(* LS UPPER TRAILING DOT 4 PHASE WINDOW *)
ls_trailing_lower_dot_4_on_comp := ls_trailing_lower_dot_4_on + less_glue_strip_deg;
ls_trailing_lower_dot_4_off_comp := ls_trailing_lower_dot_4_off - less_glue_strip_deg;

phase_window_set_phases_data(
	begin_phase:=  ls_trailing_lower_dot_4_on_comp,
	end_phase:=  ls_trailing_lower_dot_4_off_comp,
	begin_delay:= 0,
	end_delay:= 0,
	begin_max_compensation:= 0,
	end_max_compensation:= 0,
	CONVERSION_this:= ls_trailing_lower_dot_4_phwin);	

(* LS UPPER TRAILING DOT 5 PHASE WINDOW *)
ls_trailing_lower_dot_5_on_comp := ls_trailing_lower_dot_5_on + less_glue_strip_deg;
ls_trailing_lower_dot_5_off_comp := ls_trailing_lower_dot_5_off - less_glue_strip_deg;

phase_window_set_phases_data(
	begin_phase:=  ls_trailing_lower_dot_5_on_comp,
	end_phase:=  ls_trailing_lower_dot_5_off_comp,
	begin_delay:= 0,
	end_delay:= 0,
	begin_max_compensation:= 0,
	end_max_compensation:= 0,
	CONVERSION_this:= ls_trailing_lower_dot_5_phwin);
	
(* LS UPPER TRAILING DOT 6 PHASE WINDOW *)
ls_trailing_lower_dot_6_on_comp := ls_trailing_lower_dot_6_on + less_glue_strip_deg;
ls_trailing_lower_dot_6_off_comp := ls_trailing_lower_dot_6_off - less_glue_strip_deg;

phase_window_set_phases_data(
	begin_phase:=  ls_trailing_lower_dot_6_on_comp,
	end_phase:=  ls_trailing_lower_dot_6_off_comp,
	begin_delay:= 0,
	end_delay:= 0,
	begin_max_compensation:= 0,
	end_max_compensation:= 0,
	CONVERSION_this:= ls_trailing_lower_dot_6_phwin);
END_ACTION

ACTION _handle_messages:
IF purge_command
THEN 
	process_message_set(errorID_1:= 1, errorID_2:= 0, errorID_3:= 0, CONVERSION_this:= purge_running);
ELSE
	process_message_reset(purge_running);
END_IF
END_ACTION

ACTION _handle_process_test:
;
END_ACTION

ACTION _mode_manager:
IF process_mode_req_is_pending(prc)
THEN
    process_apply_mode_req_first_step(prc);
    CASE process_get_mode(prc) OF
        MODE_TO_ABSENT:
			;
        MODE_TO_INACTIVE:
			;
        MODE_TO_TEST:
			;
        MODE_TO_OPERATIONAL:
			;
    END_CASE
    process_apply_mode_req_second_step(prc);
END_IF
END_ACTION

ACTION _object_manager:
IF objects_initialization()
THEN
	sub_process_init(
		object_name					:= 'csp_case_glue.prc', 
		process						:= csp_case.prc, 
		CONVERSION_this				:= prc);
		
	prc_path 						:= process_get_path(prc);
	
	process_message_init(
		object_name:= CONCAT(prc_path, '_purge_running'), 
		behaviour:= MESSAGE_BEHAVIOUR_STATE, 
		reset_timeout:= 0, 
		disableable:= FALSE, 
		individual_reset:= FALSE, 
		machine_reaction:= MACHINE_REACTION_STOP_IN_PHASE_ONE, 
		typology:= MESSAGE_TYPOLOGY_ABNORMAL, 
		process:= prc, 
		CONVERSION_this:= purge_running);
	
	//PRS 7/14/2021	
	process_message_init(
        object_name:= CONCAT(prc_path, '_OS_lower_glue_gun_disabled_wem'),
        behaviour:= MESSAGE_BEHAVIOUR_STATE,
        reset_timeout:= 0,
        disableable:= TRUE,
        individual_reset:= FALSE,
        machine_reaction:= MACHINE_REACTION_NO_STOP, 
        typology:=  MESSAGE_TYPOLOGY_NORMAL, 
        process:= prc,
        CONVERSION_this:= OS_lower_glue_gun_disabled_wem);
	
	//PRS 7/14/2021	
	process_message_init(
        object_name:= CONCAT(prc_path, '_OS_upper_glue_gun_disabled_wem'),
        behaviour:= MESSAGE_BEHAVIOUR_STATE,
        reset_timeout:= 0,
        disableable:= TRUE,
        individual_reset:= FALSE,
        machine_reaction:= MACHINE_REACTION_NO_STOP, 
        typology:=  MESSAGE_TYPOLOGY_NORMAL, 
        process:= prc,
        CONVERSION_this:= OS_upper_glue_gun_disabled_wem);	

	//PRS 7/14/2021	
	process_message_init(
        object_name:= CONCAT(prc_path, '_LS_lower_glue_gun_disabled_wem'),
        behaviour:= MESSAGE_BEHAVIOUR_STATE,
        reset_timeout:= 0,
        disableable:= TRUE,
        individual_reset:= FALSE,
        machine_reaction:= MACHINE_REACTION_NO_STOP, 
        typology:=  MESSAGE_TYPOLOGY_NORMAL, 
        process:= prc,
        CONVERSION_this:= LS_lower_glue_gun_disabled_wem);
	
	//PRS 7/14/2021	
	process_message_init(
        object_name:= CONCAT(prc_path, '_LS_upper_glue_gun_disabled_wem'),
        behaviour:= MESSAGE_BEHAVIOUR_STATE,
        reset_timeout:= 0,
        disableable:= TRUE,
        individual_reset:= FALSE,
        machine_reaction:= MACHINE_REACTION_NO_STOP, 
        typology:=  MESSAGE_TYPOLOGY_NORMAL, 
        process:= prc,
        CONVERSION_this:= LS_upper_glue_gun_disabled_wem);		
		
		
	motorization_conditioner_init(
		object_name					:=	CONCAT(prc_path, '_purge_active_motcond'),
		velocity_limit				:=	0.0,
		velocity_limit_active		:=	FALSE,
		idle_handshake_active		:=	FALSE,
		execute_handshake_active	:=	TRUE,
		hold_handshake_active		:=	FALSE,
		suspend_handshake_active	:=	FALSE,
		complete_handshake_active	:=	FALSE,
		abort_handshake_active		:=	FALSE,
		stop_handshake_active		:=	FALSE,
		origin						:=	MOTORIZATION_CONDITIONER_ORIGIN_INTERNAL,
		manager						:=	csp_main_motorization_manager.motm,
		process						:=	prc,
		CONVERSION_this				:=	purge_active_motcond);

		
	command_button_init(
	    object_name 				:= CONCAT(prc_path, '_hmi_purge_active_cbtn'),
	    process 					:= prc,
	    CONVERSION_this 			:= hmi_purge_active_cbtn);
		
	hmi_graphic_object_status_init(
        object_name         		:= CONCAT(prc_path, '_hmi_purge_active_hgos'),
        process             		:= prc,
        CONVERSION_this             := hmi_purge_active_hgos);	
		
	hmi_graphic_object_status_init(
        object_name         		:= CONCAT(prc_path, '_hmi_glue_ready_hgos'),
        process             		:= prc,
        CONVERSION_this             := hmi_glue_ready_hgos);
		
	hmi_graphic_object_status_init(
        object_name         		:= CONCAT(prc_path, '_hmi_glue_not_ready_hgos'),
        process             		:= prc,
        CONVERSION_this             := hmi_glue_not_ready_hgos);	
	
//Glue Purge pb OS upper gun 1
	command_button_init(
	    object_name 				:= CONCAT(prc_path, '_hmi_os_glue_upper_gun1_cbtn'),
	    process 					:= prc,
	    CONVERSION_this 			:= hmi_os_glue_upper_gun1_cbtn);
		
	hmi_graphic_object_status_init(
        object_name         		:= CONCAT(prc_path, '_hmi_os_glue_upper_gun1_hgos'),
        process             		:= prc,
        CONVERSION_this             := hmi_os_glue_upper_gun1_hgos);	

//Glue Purge pb OS upper gun 2
	command_button_init(
	    object_name 				:= CONCAT(prc_path, '_hmi_os_glue_upper_gun2_cbtn'),
	    process 					:= prc,
	    CONVERSION_this 			:= hmi_os_glue_upper_gun2_cbtn);
		
	hmi_graphic_object_status_init(
        object_name         		:= CONCAT(prc_path, '_hmi_os_glue_upper_gun2_hgos'),
        process             		:= prc,
        CONVERSION_this             := hmi_os_glue_upper_gun2_hgos);			

//Glue Purge pb OS lower gun 1
	command_button_init(
	    object_name 				:= CONCAT(prc_path, '_hmi_os_glue_lower_gun1_cbtn'),
	    process 					:= prc,
	    CONVERSION_this 			:= hmi_os_glue_lower_gun1_cbtn);
		
	hmi_graphic_object_status_init(
        object_name         		:= CONCAT(prc_path, '_hmi_os_glue_lower_gun1_hgos'),
        process             		:= prc,
        CONVERSION_this             := hmi_os_glue_lower_gun1_hgos);	

//Glue Purge pb OS lower gun 2
	command_button_init(
	    object_name 				:= CONCAT(prc_path, '_hmi_os_glue_lower_gun2_cbtn'),
	    process 					:= prc,
	    CONVERSION_this 			:= hmi_os_glue_lower_gun2_cbtn);
		
	hmi_graphic_object_status_init(
        object_name         		:= CONCAT(prc_path, '_hmi_os_glue_lower_gun2_hgos'),
        process             		:= prc,
        CONVERSION_this             := hmi_os_glue_lower_gun2_hgos);	


//Glue Purge pb LS upper gun 1
	command_button_init(
	    object_name 				:= CONCAT(prc_path, '_hmi_ls_glue_upper_gun1_cbtn'),
	    process 					:= prc,
	    CONVERSION_this 			:= hmi_ls_glue_upper_gun1_cbtn);
		
	hmi_graphic_object_status_init(
        object_name         		:= CONCAT(prc_path, '_hmi_ls_glue_upper_gun1_hgos'),
        process             		:= prc,
        CONVERSION_this             := hmi_ls_glue_upper_gun1_hgos);	

//Glue Purge pb LS upper gun 2
	command_button_init(
	    object_name 				:= CONCAT(prc_path, '_hmi_ls_glue_upper_gun2_cbtn'),
	    process 					:= prc,
	    CONVERSION_this 			:= hmi_ls_glue_upper_gun2_cbtn);
		
	hmi_graphic_object_status_init(
        object_name         		:= CONCAT(prc_path, '_hmi_ls_glue_upper_gun2_hgos'),
        process             		:= prc,
        CONVERSION_this             := hmi_ls_glue_upper_gun2_hgos);			

//Glue Purge pb LS lower gun 1
	command_button_init(
	    object_name 				:= CONCAT(prc_path, '_hmi_Ls_glue_lower_gun1_cbtn'),
	    process 					:= prc,
	    CONVERSION_this 			:= hmi_ls_glue_lower_gun1_cbtn);
		
	hmi_graphic_object_status_init(
        object_name         		:= CONCAT(prc_path, '_hmi_ls_glue_lower_gun1_hgos'),
        process             		:= prc,
        CONVERSION_this             := hmi_ls_glue_lower_gun1_hgos);	

//Glue Purge pb LS lower gun 2
	command_button_init(
	    object_name 				:= CONCAT(prc_path, '_hmi_ls_glue_lower_gun2_cbtn'),
	    process 					:= prc,
	    CONVERSION_this 			:= hmi_ls_glue_lower_gun2_cbtn);
		
	hmi_graphic_object_status_init(
        object_name         		:= CONCAT(prc_path, '_hmi_ls_glue_lower_gun2_hgos'),
        process             		:= prc,
        CONVERSION_this             := hmi_ls_glue_lower_gun2_hgos);

	//Created to be the axis for the shift registers	
	phase_generator_init(
		object_name								:=CONCAT(PRC_PATH, '_glue_vm_phgen'), 
		modulo									:=360 , 
		resolution								:= PHASE_GENERATOR_RESOLUTION_UNIT, 
		axis									:= csp_case_transport_os_trailing.axis, 
		process									:=prc , 
		CONVERSION_this							:= glue_vm_phgen);

//Upper major flap check cam and phase generator		

	phase_window_init(
		object_name								:=CONCAT(PRC_PATH, '_glue_phwin'), 
		begin_phase								:=glue_leading_upper_on, 
		end_phase								:=glue_leading_upper_off, 
		begin_delay								:=0, 
		end_delay								:=0, 
		begin_max_compensation					:=0, 
		end_max_compensation					:=0, 
		generator								:=glue_vm_phgen , 
		process									:=prc , 
		CONVERSION_this							:=glue_leading_upper_phwin);	
		
//lower major flap check cam and phase generator 		

	phase_window_init(
		object_name								:=CONCAT(PRC_PATH, '_glue_phwin'), 
		begin_phase								:=glue_leading_lower_on, 
		end_phase								:=glue_leading_lower_off, 
		begin_delay								:=0, 
		end_delay								:=0, 
		begin_max_compensation					:=0, 
		end_max_compensation					:=0, 
		generator								:=glue_vm_phgen , 
		process									:=prc , 
		CONVERSION_this							:=glue_leading_lower_phwin);	

//Upper major flap check 2 cam and phase generator		
	
	phase_window_init(
		object_name								:=CONCAT(PRC_PATH, '_glue_2_phwin'), 
		begin_phase								:=glue_trailing_upper_on, 
		end_phase								:=glue_trailing_upper_off, 
		begin_delay								:=0, 
		end_delay								:=0, 
		begin_max_compensation					:=0, 
		end_max_compensation					:=0, 
		generator								:=glue_vm_phgen , 
		process									:=prc , 
		CONVERSION_this							:=glue_trailing_upper_phwin);	
		
//Lower major flap check 2 cam and phase generator		
	
	phase_window_init(
		object_name								:=CONCAT(PRC_PATH, '_glue_2_phwin'), 
		begin_phase								:=glue_trailing_lower_on, 
		end_phase								:=glue_trailing_lower_off, 
		begin_delay								:=0, 
		end_delay								:=0, 
		begin_max_compensation					:=0, 
		end_max_compensation					:=0, 
		generator								:=glue_vm_phgen , 
		process									:=prc , 
		CONVERSION_this							:=glue_trailing_lower_phwin);	
		
		
		
	(* NEW GLUE GUNS USING DIGITAL OUTPUTS *)
	digital_output_init(
		object_name 			:= CONCAT(prc_path, '_os_upper_gun_1_do'),
		polarity_direct 		:= TRUE,
		process 				:= prc,
		CONVERSION_this 		:= os_upper_gun_1_do);
		
	digital_output_init(
		object_name 			:= CONCAT(prc_path, '_os_upper_gun_2_do'),
		polarity_direct 		:= TRUE,
		process 				:= prc,
		CONVERSION_this 		:= os_upper_gun_2_do);
		
	digital_output_init(
		object_name 			:= CONCAT(prc_path, '_os_lower_gun_1_do'),
		polarity_direct 		:= TRUE,
		process 				:= prc,
		CONVERSION_this 		:= os_lower_gun_1_do);
		
	digital_output_init(
		object_name 			:= CONCAT(prc_path, '_os_lower_gun_2_do'),
		polarity_direct 		:= TRUE,
		process 				:= prc,
		CONVERSION_this 		:= os_lower_gun_2_do);
		
	digital_output_init(
		object_name 			:= CONCAT(prc_path, '_ls_upper_gun_1_do'),
		polarity_direct 		:= TRUE,
		process 				:= prc,
		CONVERSION_this 		:= ls_upper_gun_1_do);
		
	digital_output_init(
		object_name 			:= CONCAT(prc_path, '_ls_upper_gun_2_do'),
		polarity_direct 		:= TRUE,
		process 				:= prc,
		CONVERSION_this 		:= ls_upper_gun_2_do);
		
	digital_output_init(
		object_name 			:= CONCAT(prc_path, '_ls_lower_gun_1_do'),
		polarity_direct 		:= TRUE,
		process 				:= prc,
		CONVERSION_this 		:= ls_lower_gun_1_do);
		
	digital_output_init(
		object_name 			:= CONCAT(prc_path, '_ls_lower_gun_2_do'),
		polarity_direct 		:= TRUE,
		process 				:= prc,
		CONVERSION_this 		:= ls_lower_gun_2_do);
		
	(* OS LEADING UPPER PHWIN *)
	phase_window_init(
		object_name								:= CONCAT(PRC_PATH, '_os_leading_upper_dot_1_phwin'), 
		begin_phase								:= 0, // SET AT RUNTIME
		end_phase								:= 0, // SET AT RUNTIME
		begin_delay								:= 0, 
		end_delay								:= 0, 
		begin_max_compensation					:= 0, 
		end_max_compensation					:= 0, 
		generator								:= glue_vm_phgen , 
		process									:= prc , 
		CONVERSION_this							:= os_leading_upper_dot_1_phwin);	
		
	phase_window_init(
		object_name								:= CONCAT(PRC_PATH, '_os_leading_upper_dot_2_phwin'), 
		begin_phase								:= 0, // SET AT RUNTIME
		end_phase								:= 0, // SET AT RUNTIME
		begin_delay								:= 0, 
		end_delay								:= 0, 
		begin_max_compensation					:= 0, 
		end_max_compensation					:= 0, 
		generator								:= glue_vm_phgen , 
		process									:= prc , 
		CONVERSION_this							:= os_leading_upper_dot_2_phwin);	
		
	phase_window_init(
		object_name								:= CONCAT(PRC_PATH, '_os_leading_upper_dot_3_phwin'), 
		begin_phase								:= 0, // SET AT RUNTIME
		end_phase								:= 0, // SET AT RUNTIME
		begin_delay								:= 0, 
		end_delay								:= 0, 
		begin_max_compensation					:= 0, 
		end_max_compensation					:= 0, 
		generator								:= glue_vm_phgen , 
		process									:= prc , 
		CONVERSION_this							:= os_leading_upper_dot_3_phwin);	
		
	phase_window_init(
		object_name								:= CONCAT(PRC_PATH, '_os_leading_upper_dot_4_phwin'), 
		begin_phase								:= 0, // SET AT RUNTIME
		end_phase								:= 0, // SET AT RUNTIME
		begin_delay								:= 0, 
		end_delay								:= 0, 
		begin_max_compensation					:= 0, 
		end_max_compensation					:= 0, 
		generator								:= glue_vm_phgen , 
		process									:= prc , 
		CONVERSION_this							:= os_leading_upper_dot_4_phwin);	
		
	phase_window_init(
		object_name								:= CONCAT(PRC_PATH, '_os_leading_upper_dot_5_phwin'), 
		begin_phase								:= 0, // SET AT RUNTIME
		end_phase								:= 0, // SET AT RUNTIME
		begin_delay								:= 0, 
		end_delay								:= 0, 
		begin_max_compensation					:= 0, 
		end_max_compensation					:= 0, 
		generator								:= glue_vm_phgen , 
		process									:= prc , 
		CONVERSION_this							:= os_leading_upper_dot_5_phwin);	
		
	phase_window_init(
		object_name								:= CONCAT(PRC_PATH, '_os_leading_upper_dot_6_phwin'), 
		begin_phase								:= 0, // SET AT RUNTIME
		end_phase								:= 0, // SET AT RUNTIME
		begin_delay								:= 0, 
		end_delay								:= 0, 
		begin_max_compensation					:= 0, 
		end_max_compensation					:= 0, 
		generator								:= glue_vm_phgen , 
		process									:= prc , 
		CONVERSION_this							:= os_leading_upper_dot_6_phwin);
		
		
	(* OS LEADING LOWER PHWIN *)
	phase_window_init(
		object_name								:= CONCAT(PRC_PATH, '_os_leading_lower_dot_1_phwin'), 
		begin_phase								:= 0, // SET AT RUNTIME
		end_phase								:= 0, // SET AT RUNTIME
		begin_delay								:= 0, 
		end_delay								:= 0, 
		begin_max_compensation					:= 0, 
		end_max_compensation					:= 0, 
		generator								:= glue_vm_phgen , 
		process									:= prc , 
		CONVERSION_this							:= os_leading_lower_dot_1_phwin);	
		
	phase_window_init(
		object_name								:= CONCAT(PRC_PATH, '_os_leading_lower_dot_2_phwin'), 
		begin_phase								:= 0, // SET AT RUNTIME
		end_phase								:= 0, // SET AT RUNTIME
		begin_delay								:= 0, 
		end_delay								:= 0, 
		begin_max_compensation					:= 0, 
		end_max_compensation					:= 0, 
		generator								:= glue_vm_phgen , 
		process									:= prc , 
		CONVERSION_this							:= os_leading_lower_dot_2_phwin);	
		
	phase_window_init(
		object_name								:= CONCAT(PRC_PATH, '_os_leading_lower_dot_3_phwin'), 
		begin_phase								:= 0, // SET AT RUNTIME
		end_phase								:= 0, // SET AT RUNTIME
		begin_delay								:= 0, 
		end_delay								:= 0, 
		begin_max_compensation					:= 0, 
		end_max_compensation					:= 0, 
		generator								:= glue_vm_phgen , 
		process									:= prc , 
		CONVERSION_this							:= os_leading_lower_dot_3_phwin);	
		
	phase_window_init(
		object_name								:= CONCAT(PRC_PATH, '_os_leading_lower_dot_4_phwin'), 
		begin_phase								:= 0, // SET AT RUNTIME
		end_phase								:= 0, // SET AT RUNTIME
		begin_delay								:= 0, 
		end_delay								:= 0, 
		begin_max_compensation					:= 0, 
		end_max_compensation					:= 0, 
		generator								:= glue_vm_phgen , 
		process									:= prc , 
		CONVERSION_this							:= os_leading_lower_dot_4_phwin);	
		
	phase_window_init(
		object_name								:= CONCAT(PRC_PATH, '_os_leading_lower_dot_5_phwin'), 
		begin_phase								:= 0, // SET AT RUNTIME
		end_phase								:= 0, // SET AT RUNTIME
		begin_delay								:= 0, 
		end_delay								:= 0, 
		begin_max_compensation					:= 0, 
		end_max_compensation					:= 0, 
		generator								:= glue_vm_phgen , 
		process									:= prc , 
		CONVERSION_this							:= os_leading_lower_dot_5_phwin);	
		
	phase_window_init(
		object_name								:= CONCAT(PRC_PATH, '_os_leading_lower_dot_6_phwin'), 
		begin_phase								:= 0, // SET AT RUNTIME
		end_phase								:= 0, // SET AT RUNTIME
		begin_delay								:= 0, 
		end_delay								:= 0, 
		begin_max_compensation					:= 0, 
		end_max_compensation					:= 0, 
		generator								:= glue_vm_phgen , 
		process									:= prc , 
		CONVERSION_this							:= os_leading_lower_dot_6_phwin);	
		
	(* OS trailing UPPER PHWIN *)
	phase_window_init(
		object_name								:= CONCAT(PRC_PATH, '_os_trailing_upper_dot_1_phwin'), 
		begin_phase								:= 0, // SET AT RUNTIME
		end_phase								:= 0, // SET AT RUNTIME
		begin_delay								:= 0, 
		end_delay								:= 0, 
		begin_max_compensation					:= 0, 
		end_max_compensation					:= 0, 
		generator								:= glue_vm_phgen , 
		process									:= prc , 
		CONVERSION_this							:= os_trailing_upper_dot_1_phwin);	
		
	phase_window_init(
		object_name								:= CONCAT(PRC_PATH, '_os_trailing_upper_dot_2_phwin'), 
		begin_phase								:= 0, // SET AT RUNTIME
		end_phase								:= 0, // SET AT RUNTIME
		begin_delay								:= 0, 
		end_delay								:= 0, 
		begin_max_compensation					:= 0, 
		end_max_compensation					:= 0, 
		generator								:= glue_vm_phgen , 
		process									:= prc , 
		CONVERSION_this							:= os_trailing_upper_dot_2_phwin);	
		
	phase_window_init(
		object_name								:= CONCAT(PRC_PATH, '_os_trailing_upper_dot_3_phwin'), 
		begin_phase								:= 0, // SET AT RUNTIME
		end_phase								:= 0, // SET AT RUNTIME
		begin_delay								:= 0, 
		end_delay								:= 0, 
		begin_max_compensation					:= 0, 
		end_max_compensation					:= 0, 
		generator								:= glue_vm_phgen , 
		process									:= prc , 
		CONVERSION_this							:= os_trailing_upper_dot_3_phwin);	
		
	phase_window_init(
		object_name								:= CONCAT(PRC_PATH, '_os_trailing_upper_dot_4_phwin'), 
		begin_phase								:= 0, // SET AT RUNTIME
		end_phase								:= 0, // SET AT RUNTIME
		begin_delay								:= 0, 
		end_delay								:= 0, 
		begin_max_compensation					:= 0, 
		end_max_compensation					:= 0, 
		generator								:= glue_vm_phgen , 
		process									:= prc , 
		CONVERSION_this							:= os_trailing_upper_dot_4_phwin);	
		
	phase_window_init(
		object_name								:= CONCAT(PRC_PATH, '_os_trailing_upper_dot_5_phwin'), 
		begin_phase								:= 0, // SET AT RUNTIME
		end_phase								:= 0, // SET AT RUNTIME
		begin_delay								:= 0, 
		end_delay								:= 0, 
		begin_max_compensation					:= 0, 
		end_max_compensation					:= 0, 
		generator								:= glue_vm_phgen , 
		process									:= prc , 
		CONVERSION_this							:= os_trailing_upper_dot_5_phwin);	
		
	phase_window_init(
		object_name								:= CONCAT(PRC_PATH, '_os_trailing_upper_dot_6_phwin'), 
		begin_phase								:= 0, // SET AT RUNTIME
		end_phase								:= 0, // SET AT RUNTIME
		begin_delay								:= 0, 
		end_delay								:= 0, 
		begin_max_compensation					:= 0, 
		end_max_compensation					:= 0, 
		generator								:= glue_vm_phgen , 
		process									:= prc , 
		CONVERSION_this							:= os_trailing_upper_dot_6_phwin);	
		
		
	(* OS trailing LOWER PHWIN *)
	phase_window_init(
		object_name								:= CONCAT(PRC_PATH, '_os_trailing_lower_dot_1_phwin'), 
		begin_phase								:= 0, // SET AT RUNTIME
		end_phase								:= 0, // SET AT RUNTIME
		begin_delay								:= 0, 
		end_delay								:= 0, 
		begin_max_compensation					:= 0, 
		end_max_compensation					:= 0, 
		generator								:= glue_vm_phgen , 
		process									:= prc , 
		CONVERSION_this							:= os_trailing_lower_dot_1_phwin);	
		
	phase_window_init(
		object_name								:= CONCAT(PRC_PATH, '_os_trailing_lower_dot_2_phwin'), 
		begin_phase								:= 0, // SET AT RUNTIME
		end_phase								:= 0, // SET AT RUNTIME
		begin_delay								:= 0, 
		end_delay								:= 0, 
		begin_max_compensation					:= 0, 
		end_max_compensation					:= 0, 
		generator								:= glue_vm_phgen , 
		process									:= prc , 
		CONVERSION_this							:= os_trailing_lower_dot_2_phwin);	
		
	phase_window_init(
		object_name								:= CONCAT(PRC_PATH, '_os_trailing_lower_dot_3_phwin'), 
		begin_phase								:= 0, // SET AT RUNTIME
		end_phase								:= 0, // SET AT RUNTIME
		begin_delay								:= 0, 
		end_delay								:= 0, 
		begin_max_compensation					:= 0, 
		end_max_compensation					:= 0, 
		generator								:= glue_vm_phgen , 
		process									:= prc , 
		CONVERSION_this							:= os_trailing_lower_dot_3_phwin);	
		
	phase_window_init(
		object_name								:= CONCAT(PRC_PATH, '_os_trailing_lower_dot_4_phwin'), 
		begin_phase								:= 0, // SET AT RUNTIME
		end_phase								:= 0, // SET AT RUNTIME
		begin_delay								:= 0, 
		end_delay								:= 0, 
		begin_max_compensation					:= 0, 
		end_max_compensation					:= 0, 
		generator								:= glue_vm_phgen , 
		process									:= prc , 
		CONVERSION_this							:= os_trailing_lower_dot_4_phwin);
		
	phase_window_init(
		object_name								:= CONCAT(PRC_PATH, '_os_trailing_lower_dot_5_phwin'), 
		begin_phase								:= 0, // SET AT RUNTIME
		end_phase								:= 0, // SET AT RUNTIME
		begin_delay								:= 0, 
		end_delay								:= 0, 
		begin_max_compensation					:= 0, 
		end_max_compensation					:= 0, 
		generator								:= glue_vm_phgen , 
		process									:= prc , 
		CONVERSION_this							:= os_trailing_lower_dot_5_phwin);	
		
	phase_window_init(
		object_name								:= CONCAT(PRC_PATH, '_os_trailing_lower_dot_6_phwin'), 
		begin_phase								:= 0, // SET AT RUNTIME
		end_phase								:= 0, // SET AT RUNTIME
		begin_delay								:= 0, 
		end_delay								:= 0, 
		begin_max_compensation					:= 0, 
		end_max_compensation					:= 0, 
		generator								:= glue_vm_phgen , 
		process									:= prc , 
		CONVERSION_this							:= os_trailing_lower_dot_6_phwin);
		
	
	(* LS LEADING UPPER PHWIN *)
	phase_window_init(
		object_name								:= CONCAT(PRC_PATH, '_ls_leading_upper_dot_1_phwin'), 
		begin_phase								:= 0, // SET AT RUNTIME
		end_phase								:= 0, // SET AT RUNTIME
		begin_delay								:= 0, 
		end_delay								:= 0, 
		begin_max_compensation					:= 0, 
		end_max_compensation					:= 0, 
		generator								:= glue_vm_phgen , 
		process									:= prc , 
		CONVERSION_this							:= ls_leading_upper_dot_1_phwin);	
		
	phase_window_init(
		object_name								:= CONCAT(PRC_PATH, '_ls_leading_upper_dot_2_phwin'), 
		begin_phase								:= 0, // SET AT RUNTIME
		end_phase								:= 0, // SET AT RUNTIME
		begin_delay								:= 0, 
		end_delay								:= 0, 
		begin_max_compensation					:= 0, 
		end_max_compensation					:= 0, 
		generator								:= glue_vm_phgen , 
		process									:= prc , 
		CONVERSION_this							:= ls_leading_upper_dot_2_phwin);	
		
	phase_window_init(
		object_name								:= CONCAT(PRC_PATH, '_ls_leading_upper_dot_3_phwin'), 
		begin_phase								:= 0, // SET AT RUNTIME
		end_phase								:= 0, // SET AT RUNTIME
		begin_delay								:= 0, 
		end_delay								:= 0, 
		begin_max_compensation					:= 0, 
		end_max_compensation					:= 0, 
		generator								:= glue_vm_phgen , 
		process									:= prc , 
		CONVERSION_this							:= ls_leading_upper_dot_3_phwin);	
		
	phase_window_init(
		object_name								:= CONCAT(PRC_PATH, '_ls_leading_upper_dot_4_phwin'), 
		begin_phase								:= 0, // SET AT RUNTIME
		end_phase								:= 0, // SET AT RUNTIME
		begin_delay								:= 0, 
		end_delay								:= 0, 
		begin_max_compensation					:= 0, 
		end_max_compensation					:= 0, 
		generator								:= glue_vm_phgen , 
		process									:= prc , 
		CONVERSION_this							:= ls_leading_upper_dot_4_phwin);		
		
	phase_window_init(
		object_name								:= CONCAT(PRC_PATH, '_ls_leading_upper_dot_5_phwin'), 
		begin_phase								:= 0, // SET AT RUNTIME
		end_phase								:= 0, // SET AT RUNTIME
		begin_delay								:= 0, 
		end_delay								:= 0, 
		begin_max_compensation					:= 0, 
		end_max_compensation					:= 0, 
		generator								:= glue_vm_phgen , 
		process									:= prc , 
		CONVERSION_this							:= ls_leading_upper_dot_5_phwin);	
		
	phase_window_init(
		object_name								:= CONCAT(PRC_PATH, '_ls_leading_upper_dot_6_phwin'), 
		begin_phase								:= 0, // SET AT RUNTIME
		end_phase								:= 0, // SET AT RUNTIME
		begin_delay								:= 0, 
		end_delay								:= 0, 
		begin_max_compensation					:= 0, 
		end_max_compensation					:= 0, 
		generator								:= glue_vm_phgen , 
		process									:= prc , 
		CONVERSION_this							:= ls_leading_upper_dot_6_phwin);	
		
		
	(* LS LEADING LOWER PHWIN *)
	phase_window_init(
		object_name								:= CONCAT(PRC_PATH, '_ls_leading_lower_dot_1_phwin'), 
		begin_phase								:= 0, // SET AT RUNTIME
		end_phase								:= 0, // SET AT RUNTIME
		begin_delay								:= 0, 
		end_delay								:= 0, 
		begin_max_compensation					:= 0, 
		end_max_compensation					:= 0, 
		generator								:= glue_vm_phgen , 
		process									:= prc , 
		CONVERSION_this							:= ls_leading_lower_dot_1_phwin);	
		
	phase_window_init(
		object_name								:= CONCAT(PRC_PATH, '_ls_leading_lower_dot_2_phwin'), 
		begin_phase								:= 0, // SET AT RUNTIME
		end_phase								:= 0, // SET AT RUNTIME
		begin_delay								:= 0, 
		end_delay								:= 0, 
		begin_max_compensation					:= 0, 
		end_max_compensation					:= 0, 
		generator								:= glue_vm_phgen , 
		process									:= prc , 
		CONVERSION_this							:= ls_leading_lower_dot_2_phwin);	
		
	phase_window_init(
		object_name								:= CONCAT(PRC_PATH, '_ls_leading_lower_dot_3_phwin'), 
		begin_phase								:= 0, // SET AT RUNTIME
		end_phase								:= 0, // SET AT RUNTIME
		begin_delay								:= 0, 
		end_delay								:= 0, 
		begin_max_compensation					:= 0, 
		end_max_compensation					:= 0, 
		generator								:= glue_vm_phgen , 
		process									:= prc , 
		CONVERSION_this							:= ls_leading_lower_dot_3_phwin);	
		
	phase_window_init(
		object_name								:= CONCAT(PRC_PATH, '_ls_leading_lower_dot_4_phwin'), 
		begin_phase								:= 0, // SET AT RUNTIME
		end_phase								:= 0, // SET AT RUNTIME
		begin_delay								:= 0, 
		end_delay								:= 0, 
		begin_max_compensation					:= 0, 
		end_max_compensation					:= 0, 
		generator								:= glue_vm_phgen , 
		process									:= prc , 
		CONVERSION_this							:= ls_leading_lower_dot_4_phwin);		
		
	phase_window_init(
		object_name								:= CONCAT(PRC_PATH, '_ls_leading_lower_dot_5_phwin'), 
		begin_phase								:= 0, // SET AT RUNTIME
		end_phase								:= 0, // SET AT RUNTIME
		begin_delay								:= 0, 
		end_delay								:= 0, 
		begin_max_compensation					:= 0, 
		end_max_compensation					:= 0, 
		generator								:= glue_vm_phgen , 
		process									:= prc , 
		CONVERSION_this							:= ls_leading_lower_dot_5_phwin);	
		
	phase_window_init(
		object_name								:= CONCAT(PRC_PATH, '_ls_leading_lower_dot_6_phwin'), 
		begin_phase								:= 0, // SET AT RUNTIME
		end_phase								:= 0, // SET AT RUNTIME
		begin_delay								:= 0, 
		end_delay								:= 0, 
		begin_max_compensation					:= 0, 
		end_max_compensation					:= 0, 
		generator								:= glue_vm_phgen , 
		process									:= prc , 
		CONVERSION_this							:= ls_leading_lower_dot_6_phwin);	
		
	(* LS trailing UPPER PHWIN *)
	phase_window_init(
		object_name								:= CONCAT(PRC_PATH, '_ls_trailing_upper_dot_1_phwin'), 
		begin_phase								:= 0, // SET AT RUNTIME
		end_phase								:= 0, // SET AT RUNTIME
		begin_delay								:= 0, 
		end_delay								:= 0, 
		begin_max_compensation					:= 0, 
		end_max_compensation					:= 0, 
		generator								:= glue_vm_phgen , 
		process									:= prc , 
		CONVERSION_this							:= ls_trailing_upper_dot_1_phwin);	
		
	phase_window_init(
		object_name								:= CONCAT(PRC_PATH, '_ls_trailing_upper_dot_2_phwin'), 
		begin_phase								:= 0, // SET AT RUNTIME
		end_phase								:= 0, // SET AT RUNTIME
		begin_delay								:= 0, 
		end_delay								:= 0, 
		begin_max_compensation					:= 0, 
		end_max_compensation					:= 0, 
		generator								:= glue_vm_phgen , 
		process									:= prc , 
		CONVERSION_this							:= ls_trailing_upper_dot_2_phwin);	
		
	phase_window_init(
		object_name								:= CONCAT(PRC_PATH, '_ls_trailing_upper_dot_3_phwin'), 
		begin_phase								:= 0, // SET AT RUNTIME
		end_phase								:= 0, // SET AT RUNTIME
		begin_delay								:= 0, 
		end_delay								:= 0, 
		begin_max_compensation					:= 0, 
		end_max_compensation					:= 0, 
		generator								:= glue_vm_phgen , 
		process									:= prc , 
		CONVERSION_this							:= ls_trailing_upper_dot_3_phwin);	
		
	phase_window_init(
		object_name								:= CONCAT(PRC_PATH, '_ls_trailing_upper_dot_4_phwin'), 
		begin_phase								:= 0, // SET AT RUNTIME
		end_phase								:= 0, // SET AT RUNTIME
		begin_delay								:= 0, 
		end_delay								:= 0, 
		begin_max_compensation					:= 0, 
		end_max_compensation					:= 0, 
		generator								:= glue_vm_phgen , 
		process									:= prc , 
		CONVERSION_this							:= ls_trailing_upper_dot_4_phwin);	
		
	phase_window_init(
		object_name								:= CONCAT(PRC_PATH, '_ls_trailing_upper_dot_3_phwin'), 
		begin_phase								:= 0, // SET AT RUNTIME
		end_phase								:= 0, // SET AT RUNTIME
		begin_delay								:= 0, 
		end_delay								:= 0, 
		begin_max_compensation					:= 0, 
		end_max_compensation					:= 0, 
		generator								:= glue_vm_phgen , 
		process									:= prc , 
		CONVERSION_this							:= ls_trailing_upper_dot_5_phwin);	
		
	phase_window_init(
		object_name								:= CONCAT(PRC_PATH, '_ls_trailing_upper_dot_4_phwin'), 
		begin_phase								:= 0, // SET AT RUNTIME
		end_phase								:= 0, // SET AT RUNTIME
		begin_delay								:= 0, 
		end_delay								:= 0, 
		begin_max_compensation					:= 0, 
		end_max_compensation					:= 0, 
		generator								:= glue_vm_phgen , 
		process									:= prc , 
		CONVERSION_this							:= ls_trailing_upper_dot_6_phwin);	
		
		
	(* LS trailing LOWER PHWIN *)
	phase_window_init(
		object_name								:= CONCAT(PRC_PATH, '_ls_trailing_lower_dot_1_phwin'), 
		begin_phase								:= 0, // SET AT RUNTIME
		end_phase								:= 0, // SET AT RUNTIME
		begin_delay								:= 0, 
		end_delay								:= 0, 
		begin_max_compensation					:= 0, 
		end_max_compensation					:= 0, 
		generator								:= glue_vm_phgen , 
		process									:= prc , 
		CONVERSION_this							:= ls_trailing_lower_dot_1_phwin);	
		
	phase_window_init(
		object_name								:= CONCAT(PRC_PATH, '_ls_trailing_lower_dot_2_phwin'), 
		begin_phase								:= 0, // SET AT RUNTIME
		end_phase								:= 0, // SET AT RUNTIME
		begin_delay								:= 0, 
		end_delay								:= 0, 
		begin_max_compensation					:= 0, 
		end_max_compensation					:= 0, 
		generator								:= glue_vm_phgen , 
		process									:= prc , 
		CONVERSION_this							:= ls_trailing_lower_dot_2_phwin);	
		
	phase_window_init(
		object_name								:= CONCAT(PRC_PATH, '_ls_trailing_lower_dot_3_phwin'), 
		begin_phase								:= 0, // SET AT RUNTIME
		end_phase								:= 0, // SET AT RUNTIME
		begin_delay								:= 0, 
		end_delay								:= 0, 
		begin_max_compensation					:= 0, 
		end_max_compensation					:= 0, 
		generator								:= glue_vm_phgen , 
		process									:= prc , 
		CONVERSION_this							:= ls_trailing_lower_dot_3_phwin);	
		
	phase_window_init(
		object_name								:= CONCAT(PRC_PATH, '_ls_trailing_lower_dot_4_phwin'), 
		begin_phase								:= 0, // SET AT RUNTIME
		end_phase								:= 0, // SET AT RUNTIME
		begin_delay								:= 0, 
		end_delay								:= 0, 
		begin_max_compensation					:= 0, 
		end_max_compensation					:= 0, 
		generator								:= glue_vm_phgen , 
		process									:= prc , 
		CONVERSION_this							:= ls_trailing_lower_dot_4_phwin);
		
	phase_window_init(
		object_name								:= CONCAT(PRC_PATH, '_ls_trailing_lower_dot_3_phwin'), 
		begin_phase								:= 0, // SET AT RUNTIME
		end_phase								:= 0, // SET AT RUNTIME
		begin_delay								:= 0, 
		end_delay								:= 0, 
		begin_max_compensation					:= 0, 
		end_max_compensation					:= 0, 
		generator								:= glue_vm_phgen , 
		process									:= prc , 
		CONVERSION_this							:= ls_trailing_lower_dot_5_phwin);	
		
	phase_window_init(
		object_name								:= CONCAT(PRC_PATH, '_ls_trailing_lower_dot_4_phwin'), 
		begin_phase								:= 0, // SET AT RUNTIME
		end_phase								:= 0, // SET AT RUNTIME
		begin_delay								:= 0, 
		end_delay								:= 0, 
		begin_max_compensation					:= 0, 
		end_max_compensation					:= 0, 
		generator								:= glue_vm_phgen , 
		process									:= prc , 
		CONVERSION_this							:= ls_trailing_lower_dot_6_phwin);
		
		
	(* GUN DO TIMER ON TIMEOUTS *)
	timer_init(
		object_name					:= CONCAT(prc_path, '_os_upper_gun_1_on_tmr'),
		process						:= prc,
		CONVERSION_this				:= os_upper_gun_1_on_tmr);
		
	timer_init(
		object_name					:= CONCAT(prc_path, '_os_upper_gun_2_on_tmr'),
		process						:= prc,
		CONVERSION_this				:= os_upper_gun_2_on_tmr);
		
	timer_init(
		object_name					:= CONCAT(prc_path, '_os_lower_gun_1_on_tmr'),
		process						:= prc,
		CONVERSION_this				:= os_lower_gun_1_on_tmr);
		
	timer_init(
		object_name					:= CONCAT(prc_path, '_os_lower_gun_2_on_tmr'),
		process						:= prc,
		CONVERSION_this				:= os_lower_gun_2_on_tmr);
		
	
	timer_init(
		object_name					:= CONCAT(prc_path, '_ls_upper_gun_1_on_tmr'),
		process						:= prc,
		CONVERSION_this				:= ls_upper_gun_1_on_tmr);
		
	timer_init(
		object_name					:= CONCAT(prc_path, '_ls_upper_gun_2_on_tmr'),
		process						:= prc,
		CONVERSION_this				:= ls_upper_gun_2_on_tmr);
		
	timer_init(
		object_name					:= CONCAT(prc_path, '_ls_lower_gun_1_on_tmr'),
		process						:= prc,
		CONVERSION_this				:= ls_lower_gun_1_on_tmr);
		
	timer_init(
		object_name					:= CONCAT(prc_path, '_ls_lower_gun_2_on_tmr'),
		process						:= prc,
		CONVERSION_this				:= ls_lower_gun_2_on_tmr);	

END_IF

IF objects_running()
THEN
	process_cycle(prc);
	phase_generator_cycle(glue_vm_phgen);
	motorization_conditioner_cycle(purge_active_motcond);
	
	phase_window_cycle(glue_leading_upper_phwin);
	phase_window_cycle(glue_trailing_upper_phwin);
	phase_window_cycle(glue_leading_lower_phwin);
	phase_window_cycle(glue_trailing_lower_phwin);
	
	command_button_cycle(hmi_purge_active_cbtn);
	command_button_cycle(hmi_os_glue_upper_gun1_cbtn);
	command_button_cycle(hmi_os_glue_upper_gun2_cbtn);
	command_button_cycle(hmi_os_glue_lower_gun1_cbtn);
	command_button_cycle(hmi_os_glue_lower_gun2_cbtn);
	command_button_cycle(hmi_ls_glue_upper_gun1_cbtn);
	command_button_cycle(hmi_ls_glue_upper_gun2_cbtn);
	command_button_cycle(hmi_ls_glue_lower_gun1_cbtn);
	command_button_cycle(hmi_ls_glue_lower_gun2_cbtn);
	
	(* NEW OUTPUT PHWIN *)
	
	(* OS PHWIN *)
	phase_window_cycle(os_leading_upper_dot_1_phwin);
	phase_window_cycle(os_leading_upper_dot_2_phwin);
	phase_window_cycle(os_leading_upper_dot_3_phwin);
	phase_window_cycle(os_leading_upper_dot_4_phwin);
	phase_window_cycle(os_leading_upper_dot_5_phwin);
	phase_window_cycle(os_leading_upper_dot_6_phwin);
	
	phase_window_cycle(os_leading_lower_dot_1_phwin);
	phase_window_cycle(os_leading_lower_dot_2_phwin);
	phase_window_cycle(os_leading_lower_dot_3_phwin);
	phase_window_cycle(os_leading_lower_dot_4_phwin);
	phase_window_cycle(os_leading_lower_dot_5_phwin);
	phase_window_cycle(os_leading_lower_dot_6_phwin);
	
	phase_window_cycle(os_trailing_upper_dot_1_phwin);
	phase_window_cycle(os_trailing_upper_dot_2_phwin);
	phase_window_cycle(os_trailing_upper_dot_3_phwin);
	phase_window_cycle(os_trailing_upper_dot_4_phwin);
	phase_window_cycle(os_trailing_upper_dot_5_phwin);
	phase_window_cycle(os_trailing_upper_dot_6_phwin);
	
	phase_window_cycle(os_trailing_lower_dot_1_phwin);
	phase_window_cycle(os_trailing_lower_dot_2_phwin);
	phase_window_cycle(os_trailing_lower_dot_3_phwin);
	phase_window_cycle(os_trailing_lower_dot_4_phwin);
	phase_window_cycle(os_trailing_lower_dot_5_phwin);
	phase_window_cycle(os_trailing_lower_dot_6_phwin);
	
	(* LS PHWIN *)
	phase_window_cycle(ls_leading_upper_dot_1_phwin);
	phase_window_cycle(ls_leading_upper_dot_2_phwin);
	phase_window_cycle(ls_leading_upper_dot_3_phwin);
	phase_window_cycle(ls_leading_upper_dot_4_phwin);
	phase_window_cycle(ls_leading_upper_dot_5_phwin);
	phase_window_cycle(ls_leading_upper_dot_6_phwin);
	
	phase_window_cycle(ls_leading_lower_dot_1_phwin);
	phase_window_cycle(ls_leading_lower_dot_2_phwin);
	phase_window_cycle(ls_leading_lower_dot_3_phwin);
	phase_window_cycle(ls_leading_lower_dot_4_phwin);
	phase_window_cycle(ls_leading_lower_dot_5_phwin);
	phase_window_cycle(ls_leading_lower_dot_6_phwin);
	
	phase_window_cycle(ls_trailing_upper_dot_1_phwin);
	phase_window_cycle(ls_trailing_upper_dot_2_phwin);
	phase_window_cycle(ls_trailing_upper_dot_3_phwin);
	phase_window_cycle(ls_trailing_upper_dot_4_phwin);
	phase_window_cycle(ls_trailing_upper_dot_5_phwin);
	phase_window_cycle(ls_trailing_upper_dot_6_phwin);
	
	phase_window_cycle(ls_trailing_lower_dot_1_phwin);
	phase_window_cycle(ls_trailing_lower_dot_2_phwin);
	phase_window_cycle(ls_trailing_lower_dot_3_phwin);
	phase_window_cycle(ls_trailing_lower_dot_4_phwin);
	phase_window_cycle(ls_trailing_lower_dot_5_phwin);
	phase_window_cycle(ls_trailing_lower_dot_6_phwin);
	
END_IF
END_ACTION

ACTION _read_process_image:
;
END_ACTION

ACTION _read_var_input:
;
END_ACTION

ACTION _run_cycle_NEW:
enable_conditions :=
	digital_input_is_active(csp_case_glue_hotMelt.ready_di);	

(* GLUE IS READY AND MACHINE IS STOPPED READY FOR PURGE *)
IF	enable_conditions
	AND
	(	
		motorization_manager_is_stopped(csp_main_motorization_manager.motm)
		OR
		motorization_manager_is_aborted(csp_main_motorization_manager.motm)
	)
THEN
	(* Purge HMI Button enable - LINKED TO HMI *)
	IF purge_req	
	THEN
		(* At the moment there not purge position as well as Cartoner !! *)
		purge_position := TRUE;
		run_position := FALSE;
	ELSE
		purge_position := FALSE;
		run_position := TRUE;	
	END_IF
END_IF

	
purge_conditions :=
	enable_conditions
	AND
	purge_req;
	//AND
	//purge_position;
	
run_conditions :=
	enable_conditions (* GLUE HOTMELT IS READY *)
	AND csp_main_motorization_virtualManager.axis.actual_velocity > 0 (* MAIN MOTORIZATION IS MOVING *)
	AND NOT hot_glue_bypass;
	

CASE fsm_status_NEW OF
	
	(* CHECKS TO SEE IF IT WILL BE PURGE OR RUN *)
	CSP_CASE_GLUE_STATUS_INIT:
	
		purge_in_progress := FALSE;
	
		IF purge_conditions
		THEN
			purge_in_progress := TRUE;
			fsm_next_status_NEW := CSP_CASE_GLUE_STATUS_PURGE_ACTIVATE;
		ELSIF run_conditions
		THEN	
			fsm_next_status_NEW := CSP_CASE_GLUE_STATUS_RUNNING;
		END_IF
		
		
	(* PURGE ACTIVATE *)
	CSP_CASE_GLUE_STATUS_PURGE_ACTIVATE:
	
		(* OS UPPER GUN 1 *)
		IF	command_button_is_pressed(hmi_os_glue_upper_gun1_cbtn)  
		THEN
			digital_output_set(os_upper_gun_1_do);
		ELSE
			digital_output_reset(os_upper_gun_1_do);
		END_IF
		
		(* OS UPPER GUN 2 *)
		IF	command_button_is_pressed(hmi_os_glue_upper_gun2_cbtn)  
		THEN
			digital_output_set(os_upper_gun_2_do);
		ELSE
			digital_output_reset(os_upper_gun_2_do);
		END_IF
		
		(* OS LOWER GUN 1 *)
		IF	command_button_is_pressed(hmi_os_glue_lower_gun1_cbtn)  
		THEN
			digital_output_set(os_lower_gun_1_do);
		ELSE
			digital_output_reset(os_lower_gun_1_do);
		END_IF
		
		(* OS LOWER GUN 2 *)
		IF	command_button_is_pressed(hmi_os_glue_lower_gun2_cbtn) 
		THEN
			digital_output_set(os_lower_gun_2_do);
		ELSE
			digital_output_reset(os_lower_gun_2_do);
		END_IF
		
		(* LS UPPER GUN 1 *)
		IF	command_button_is_pressed(hmi_ls_glue_upper_gun1_cbtn)  
		THEN
			digital_output_set(ls_upper_gun_1_do);
		ELSE
			digital_output_reset(ls_upper_gun_1_do);
		END_IF
		
		(* LS UPPER GUN 2 *)
		IF	command_button_is_pressed(hmi_ls_glue_upper_gun2_cbtn) 
		THEN
			digital_output_set(ls_upper_gun_2_do);
		ELSE
			digital_output_reset(ls_upper_gun_2_do);
		END_IF
		
		(* LS LOWER GUN 1 *)
		IF	command_button_is_pressed(hmi_ls_glue_lower_gun1_cbtn) 
		THEN
			digital_output_set(ls_lower_gun_1_do);
		ELSE
			digital_output_reset(ls_lower_gun_1_do);
		END_IF
		
		(* LS LOWER GUN 2 *)
		IF	command_button_is_pressed(hmi_ls_glue_lower_gun2_cbtn) 
		THEN
			digital_output_set(ls_lower_gun_2_do);
		ELSE
			digital_output_reset(ls_lower_gun_2_do);
		END_IF
		
		
		IF NOT purge_conditions
		THEN
			fsm_next_status_NEW := CSP_CASE_GLUE_STATUS_PURGE_WAITING_DEACTIVATE;
		END_IF
		
		
	(* RESET ALL GLUE DIGITAL OUTPUTS *)
	CSP_CASE_GLUE_STATUS_PURGE_WAITING_DEACTIVATE:
		
		(* OS GUNS RESET *)
		digital_output_reset(os_upper_gun_1_do);
		digital_output_reset(os_upper_gun_2_do);
		digital_output_reset(os_lower_gun_1_do);
		digital_output_reset(os_lower_gun_2_do);
		
		(* LS GUNS RESET *)
		digital_output_reset(ls_upper_gun_1_do);
		digital_output_reset(ls_upper_gun_2_do);
		digital_output_reset(ls_lower_gun_1_do);
		digital_output_reset(ls_lower_gun_2_do);
		
		fsm_next_status_NEW := CSP_CASE_GLUE_STATUS_INIT;		
	
		
	(* RUNNING CONDITIONS ARE MET - MACHINE IS IN RUN MODE *)	
	CSP_CASE_GLUE_STATUS_RUNNING:

		(* OS GLUE PE GOES HIGH AND TRAILING LUG IS MOVING - CASE AT GLUE LATCH *)
		IF digital_input_is_active(csp_case_glue_sensors.case_present_os_di) 
			AND digital_input_is_active(csp_case_glue_sensors.case_present_ls_di) 
			AND axis_is_moving(csp_case_transport_os_trailing.axis)
			AND axis_is_cam_engaged(csp_case_transport_os_trailing.axis)
		THEN
			os_case_at_glue_latch := TRUE;
		END_IF
		
		(* LS GLUE PE GOES HIGH AND TRAILING LUG IS MOVING - CASE AT GLUE LATCH *)
		IF digital_input_is_active(csp_case_glue_sensors.case_present_ls_di) 
			AND digital_input_is_active(csp_case_glue_sensors.case_present_os_di) 
			AND axis_is_moving(csp_case_transport_os_trailing.axis)
			AND axis_is_cam_engaged(csp_case_transport_os_trailing.axis)
		THEN
			ls_case_at_glue_latch := TRUE;
		END_IF
		
		
		(* CASE AT GLUE GOES FALSE WHEN AXIS IS MOVING AND MODULO GOES OUT OF RANGE *)
		IF (os_case_at_glue_latch OR ls_case_at_glue_latch)
			AND axis_is_moving(csp_case_transport_os_trailing.axis) 
			AND axis_get_actual_modulo_position(csp_case_transport_os_trailing.axis) > glue_trailing_upper_off //unlatch case at glue when past trailing glue flap window
			OR NOT axis_is_cam_engaged(csp_case_transport_os_trailing.axis)
			OR (csp.o_machine_is_stopped
			AND NOT axis_is_moving(csp_case_virtualMaster.axis))//unlatch on stop since glue will dry before closing
		THEN
			os_case_at_glue_latch := FALSE;
			ls_case_at_glue_latch := FALSE;
		END_IF
		
		IF toggle_shift_reg 
			AND	
			shift_register_step_has_status_item(
			step_id := case_at_glue_sr,
			status_bits_to_be_true := ITEM_HAS_LOAD,
			status_bits_to_be_false := 0,
			CONVERSION_this :=csp_case_main_statistics.sr)
		THEN 
			glue_shift_active :=TRUE;
		ELSE
			glue_shift_active :=FALSE;
		END_IF				
	
		
	(* RUN CONDITIONS *)
		IF run_conditions
			AND axis_is_moving(csp_case_transport_os_trailing.axis)
		THEN
			(* CHECKS PHASE WINDOWS TO DETERMINE IF GLUE GUN SHOULD BE ON *)
			
			(* OS UPPER DOTS *)
			IF os_case_at_glue_latch
				AND (
						(dot_1_enable AND phase_window_position_is_in_window(axis_get_actual_modulo_position(csp_case_transport_os_trailing.axis), os_leading_upper_dot_1_phwin)) (* LEADING UPPER DOT 1 *)
						OR (dot_2_enable AND phase_window_position_is_in_window(axis_get_actual_modulo_position(csp_case_transport_os_trailing.axis), os_leading_upper_dot_2_phwin)) (* LEADING UPPER DOT 2 *)
						OR (dot_3_enable AND phase_window_position_is_in_window(axis_get_actual_modulo_position(csp_case_transport_os_trailing.axis), os_leading_upper_dot_3_phwin)) (* LEADING UPPER DOT 3 *)
						OR (dot_4_enable AND phase_window_position_is_in_window(axis_get_actual_modulo_position(csp_case_transport_os_trailing.axis), os_leading_upper_dot_4_phwin)) (* LEADING UPPER DOT 4 *)
						OR (dot_5_enable AND phase_window_position_is_in_window(axis_get_actual_modulo_position(csp_case_transport_os_trailing.axis), os_leading_upper_dot_5_phwin)) (* LEADING UPPER DOT 5 *)
						OR (dot_6_enable AND phase_window_position_is_in_window(axis_get_actual_modulo_position(csp_case_transport_os_trailing.axis), os_leading_upper_dot_6_phwin)) (* LEADING UPPER DOT 6 *)
						OR (dot_1_enable AND phase_window_position_is_in_window(axis_get_actual_modulo_position(csp_case_transport_os_trailing.axis), os_trailing_upper_dot_1_phwin)) (* TRAILING UPPER DOT 1 *)
						OR (dot_2_enable AND phase_window_position_is_in_window(axis_get_actual_modulo_position(csp_case_transport_os_trailing.axis), os_trailing_upper_dot_2_phwin)) (* TRAILING UPPER DOT 2 *)
						OR (dot_3_enable AND phase_window_position_is_in_window(axis_get_actual_modulo_position(csp_case_transport_os_trailing.axis), os_trailing_upper_dot_3_phwin)) (* TRAILING UPPER DOT 3 *)
						OR (dot_4_enable AND phase_window_position_is_in_window(axis_get_actual_modulo_position(csp_case_transport_os_trailing.axis), os_trailing_upper_dot_4_phwin)) (* TRAILING UPPER DOT 4 *)
						OR (dot_5_enable AND phase_window_position_is_in_window(axis_get_actual_modulo_position(csp_case_transport_os_trailing.axis), os_trailing_upper_dot_5_phwin)) (* TRAILING UPPER DOT 5 *)
						OR (dot_6_enable AND phase_window_position_is_in_window(axis_get_actual_modulo_position(csp_case_transport_os_trailing.axis), os_trailing_upper_dot_6_phwin)) (* TRAILING UPPER DOT 6 *)
				)
				AND NOT os_upper_bypass_req
			THEN
					(* OS UPPER GUN 1 IF ENABLED *)
					IF os_upper_gun_1_enable
					THEN
						digital_output_set(os_upper_gun_1_do);
					END_IF
					(* OS UPPER GUN 2 IF ENABLED *)
					IF os_upper_gun_2_enable
					THEN
						digital_output_set(os_upper_gun_2_do);
					END_IF
			ELSE
				digital_output_reset(os_upper_gun_1_do);
				digital_output_reset(os_upper_gun_2_do);
			END_IF
			
			(* OS LOWER DOTS *)
			IF os_case_at_glue_latch
				AND (
						(dot_1_enable AND phase_window_position_is_in_window(axis_get_actual_modulo_position(csp_case_transport_os_trailing.axis), os_leading_lower_dot_1_phwin)) (* LEADING lower DOT 1 *)
						OR (dot_2_enable AND phase_window_position_is_in_window(axis_get_actual_modulo_position(csp_case_transport_os_trailing.axis), os_leading_lower_dot_2_phwin)) (* LEADING lower DOT 2 *)
						OR (dot_3_enable AND phase_window_position_is_in_window(axis_get_actual_modulo_position(csp_case_transport_os_trailing.axis), os_leading_lower_dot_3_phwin)) (* LEADING lower DOT 3 *)
						OR (dot_4_enable AND phase_window_position_is_in_window(axis_get_actual_modulo_position(csp_case_transport_os_trailing.axis), os_leading_lower_dot_4_phwin)) (* LEADING lower DOT 4 *)
						OR (dot_5_enable AND phase_window_position_is_in_window(axis_get_actual_modulo_position(csp_case_transport_os_trailing.axis), os_leading_lower_dot_5_phwin)) (* LEADING lower DOT 5 *)
						OR (dot_6_enable AND phase_window_position_is_in_window(axis_get_actual_modulo_position(csp_case_transport_os_trailing.axis), os_leading_lower_dot_6_phwin)) (* LEADING lower DOT 6 *)
						OR (dot_1_enable AND phase_window_position_is_in_window(axis_get_actual_modulo_position(csp_case_transport_os_trailing.axis), os_trailing_lower_dot_1_phwin)) (* TRAILING lower DOT 1 *)
						OR (dot_2_enable AND phase_window_position_is_in_window(axis_get_actual_modulo_position(csp_case_transport_os_trailing.axis), os_trailing_lower_dot_2_phwin)) (* TRAILING lower DOT 2 *)
						OR (dot_3_enable AND phase_window_position_is_in_window(axis_get_actual_modulo_position(csp_case_transport_os_trailing.axis), os_trailing_lower_dot_3_phwin)) (* TRAILING lower DOT 3 *)
						OR (dot_4_enable AND phase_window_position_is_in_window(axis_get_actual_modulo_position(csp_case_transport_os_trailing.axis), os_trailing_lower_dot_4_phwin)) (* TRAILING lower DOT 4 *)
						OR (dot_5_enable AND phase_window_position_is_in_window(axis_get_actual_modulo_position(csp_case_transport_os_trailing.axis), os_trailing_lower_dot_5_phwin)) (* TRAILING lower DOT 5 *)
						OR (dot_6_enable AND phase_window_position_is_in_window(axis_get_actual_modulo_position(csp_case_transport_os_trailing.axis), os_trailing_lower_dot_6_phwin)) (* TRAILING lower DOT 6 *)
				)
				AND NOT os_lower_bypass_req
			THEN
				(* OS LOWER GUN 1 IF ENABLED *)
				IF os_lower_gun_1_enable
				THEN
					digital_output_set(os_lower_gun_1_do);
				END_IF
				(* OS LOWER GUN 2 IF ENABLED *)
				IF os_lower_gun_2_enable
				THEN
					digital_output_set(os_lower_gun_2_do);
				END_IF
			ELSE
				digital_output_reset(os_lower_gun_1_do);
				digital_output_reset(os_lower_gun_2_do);
			END_IF
			
			
			(* LS UPPER DOTS *)
			IF ls_case_at_glue_latch
				AND (
						(dot_1_enable AND phase_window_position_is_in_window(axis_get_actual_modulo_position(csp_case_transport_ls_trailing.axis), ls_leading_upper_dot_1_phwin)) (* LEADING UPPER DOT 1 *)
						OR (dot_2_enable AND phase_window_position_is_in_window(axis_get_actual_modulo_position(csp_case_transport_ls_trailing.axis), ls_leading_upper_dot_2_phwin)) (* LEADING UPPER DOT 2 *)
						OR (dot_3_enable AND phase_window_position_is_in_window(axis_get_actual_modulo_position(csp_case_transport_ls_trailing.axis), ls_leading_upper_dot_3_phwin)) (* LEADING UPPER DOT 3 *)
						OR (dot_4_enable AND phase_window_position_is_in_window(axis_get_actual_modulo_position(csp_case_transport_ls_trailing.axis), ls_leading_upper_dot_4_phwin)) (* LEADING UPPER DOT 4 *)
						OR (dot_5_enable AND phase_window_position_is_in_window(axis_get_actual_modulo_position(csp_case_transport_ls_trailing.axis), ls_leading_upper_dot_5_phwin)) (* LEADING UPPER DOT 5 *)
						OR (dot_6_enable AND phase_window_position_is_in_window(axis_get_actual_modulo_position(csp_case_transport_ls_trailing.axis), ls_leading_upper_dot_6_phwin)) (* LEADING UPPER DOT 6 *)
						OR (dot_1_enable AND phase_window_position_is_in_window(axis_get_actual_modulo_position(csp_case_transport_ls_trailing.axis), ls_trailing_upper_dot_1_phwin)) (* TRAILING UPPER DOT 1 *)
						OR (dot_2_enable AND phase_window_position_is_in_window(axis_get_actual_modulo_position(csp_case_transport_ls_trailing.axis), ls_trailing_upper_dot_2_phwin)) (* TRAILING UPPER DOT 2 *)
						OR (dot_3_enable AND phase_window_position_is_in_window(axis_get_actual_modulo_position(csp_case_transport_ls_trailing.axis), ls_trailing_upper_dot_3_phwin)) (* TRAILING UPPER DOT 3 *)
						OR (dot_4_enable AND phase_window_position_is_in_window(axis_get_actual_modulo_position(csp_case_transport_ls_trailing.axis), ls_trailing_upper_dot_4_phwin)) (* TRAILING UPPER DOT 4 *)
						OR (dot_5_enable AND phase_window_position_is_in_window(axis_get_actual_modulo_position(csp_case_transport_ls_trailing.axis), ls_trailing_upper_dot_5_phwin)) (* TRAILING UPPER DOT 3 *)
						OR (dot_6_enable AND phase_window_position_is_in_window(axis_get_actual_modulo_position(csp_case_transport_ls_trailing.axis), ls_trailing_upper_dot_6_phwin)) (* TRAILING UPPER DOT 4 *)
				)
				AND NOT ls_upper_bypass_req
			THEN
				(* LS UPPER GUN 1 IF ENABLED *)
				IF ls_upper_gun_1_enable
				THEN
					digital_output_set(ls_upper_gun_1_do);
				END_IF
				(* LS UPPER GUN 2 IF ENABLED *)
				IF ls_upper_gun_2_enable
				THEN
					digital_output_set(ls_upper_gun_2_do);
				END_IF
			ELSE
				digital_output_reset(ls_upper_gun_1_do);
				digital_output_reset(ls_upper_gun_2_do);
			END_IF
			
			(* LS LOWER DOTS *)
			IF ls_case_at_glue_latch
				AND (
						(dot_1_enable AND phase_window_position_is_in_window(axis_get_actual_modulo_position(csp_case_transport_ls_trailing.axis), ls_leading_lower_dot_1_phwin)) (* LEADING lower DOT 1 *)
						OR (dot_2_enable AND phase_window_position_is_in_window(axis_get_actual_modulo_position(csp_case_transport_ls_trailing.axis), ls_leading_lower_dot_2_phwin)) (* LEADING lower DOT 2 *)
						OR (dot_3_enable AND phase_window_position_is_in_window(axis_get_actual_modulo_position(csp_case_transport_ls_trailing.axis), ls_leading_lower_dot_3_phwin)) (* LEADING lower DOT 3 *)
						OR (dot_4_enable AND phase_window_position_is_in_window(axis_get_actual_modulo_position(csp_case_transport_ls_trailing.axis), ls_leading_lower_dot_4_phwin)) (* LEADING lower DOT 4 *)
						OR (dot_5_enable AND phase_window_position_is_in_window(axis_get_actual_modulo_position(csp_case_transport_ls_trailing.axis), ls_leading_lower_dot_5_phwin)) (* LEADING lower DOT 5 *)
						OR (dot_6_enable AND phase_window_position_is_in_window(axis_get_actual_modulo_position(csp_case_transport_ls_trailing.axis), ls_leading_lower_dot_6_phwin)) (* LEADING lower DOT 6 *)
						OR (dot_1_enable AND phase_window_position_is_in_window(axis_get_actual_modulo_position(csp_case_transport_ls_trailing.axis), ls_trailing_lower_dot_1_phwin)) (* TRAILING lower DOT 1 *)
						OR (dot_2_enable AND phase_window_position_is_in_window(axis_get_actual_modulo_position(csp_case_transport_ls_trailing.axis), ls_trailing_lower_dot_2_phwin)) (* TRAILING lower DOT 2 *)
						OR (dot_3_enable AND phase_window_position_is_in_window(axis_get_actual_modulo_position(csp_case_transport_ls_trailing.axis), ls_trailing_lower_dot_3_phwin)) (* TRAILING lower DOT 3 *)
						OR (dot_4_enable AND phase_window_position_is_in_window(axis_get_actual_modulo_position(csp_case_transport_ls_trailing.axis), ls_trailing_lower_dot_4_phwin)) (* TRAILING lower DOT 4 *)
						OR (dot_5_enable AND phase_window_position_is_in_window(axis_get_actual_modulo_position(csp_case_transport_ls_trailing.axis), ls_trailing_lower_dot_5_phwin)) (* TRAILING lower DOT 3 *)
						OR (dot_6_enable AND phase_window_position_is_in_window(axis_get_actual_modulo_position(csp_case_transport_ls_trailing.axis), ls_trailing_lower_dot_6_phwin)) (* TRAILING lower DOT 4 *)
				)
				AND NOT ls_lower_bypass_req
			THEN
				(* LS LOWER GUN 1 IF ENABLED *)
				IF ls_lower_gun_1_enable
				THEN
					digital_output_set(ls_lower_gun_1_do);
				END_IF
				(* LS LOWER GUN 2 IF ENABLED *)
				IF ls_lower_gun_2_enable
				THEN
					digital_output_set(ls_lower_gun_2_do);
				END_IF
			ELSE
				digital_output_reset(ls_lower_gun_1_do);
				digital_output_reset(ls_lower_gun_2_do);
			END_IF
			
			
		ELSE (* LOST RUN CONDITIONS OR GLUE LATCH OR AXIS IS NOT MOVING *)
			(* OS GUNS RESET *)
			digital_output_reset(os_upper_gun_1_do);
			digital_output_reset(os_upper_gun_2_do);
			digital_output_reset(os_lower_gun_1_do);
			digital_output_reset(os_lower_gun_2_do);
			
			(* LS GUNS RESET *)
			digital_output_reset(ls_upper_gun_1_do);
			digital_output_reset(ls_upper_gun_2_do);
			digital_output_reset(ls_lower_gun_1_do);
			digital_output_reset(ls_lower_gun_2_do);
			
			fsm_next_status_NEW := CSP_CASE_GLUE_STATUS_INIT;
		END_IF
				
END_CASE


IF NOT debug_state_machine
	OR
	debug_state_machine_one_step
THEN
	fsm_status_NEW := fsm_next_status_NEW; // TEMP RMH 9.16.2020
	debug_state_machine_one_step := FALSE;
END_IF
END_ACTION

ACTION _set_runtime_properties:
;
END_ACTION

ACTION _write_output:
;
END_ACTION

END_PROGRAM

// ---- Application/CSP/Case/Glue/Sensors/csp_case_glue_sensors.TcPOU
(*********************************** G.D S.p.A. - Technical Department ***********************************
============= PROGRAM INFO ============
FOLDER:             TBD
MACHINES INVOLVED:  TBD 

============= DESCRIPTION =============
csp machine declaration

============= REVISIONS ===============
Date		Version	 	Author      	Description             
----------	-------		------------  	--------------------------------------------
2019/04/05 	0000.00	 	M.Grasso		Creation of the PRG

**********************************************************************************************************)
(*$R process_ref := prc; $*)
PROGRAM csp_case_glue_sensors
VAR
	
	prc:											process;
	prc_path:										STRING;
	
	case_present_os_di:								digital_input;
	case_present_os_di_dchk: 						check_section;
	
	
	case_present_ls_di:								digital_input;
	case_present_ls_di_dchk: 						check_section;
	
	Case_at_glue_begin_phase:						LREAL:=150;
	Case_at_glue_end_phase:							LREAL:=180;
	
	bad_count_os: 									INT;
	consecutive_blocked_os_aem:						message;
	consecutive_blocked_ls_aem:						message;
	bad_count_ls: 									INT;
	temp1: 											BOOL;
	temp2: 											BOOL;
	consecutive_blocked_count:						INT := 3;
END_VAR

_read_var_input();

_object_manager();

IF NOT objects_running()
THEN
	RETURN;	
END_IF

_read_process_image();

_mode_manager();

_set_runtime_properties();

(********************************* BODY *********************************)
check_section_set_check_window_phases_value(
    begin_phase         :=  Case_at_glue_begin_phase,
    end_phase           :=  Case_at_glue_end_phase,
    conversion_THIS     :=  case_present_os_di_dchk);	
	
check_section_set_check_window_phases_value(
    begin_phase         :=  Case_at_glue_begin_phase,
    end_phase           :=  Case_at_glue_end_phase,
    conversion_THIS     :=  case_present_ls_di_dchk);	

(* TRACKS IF PE WAS BAD DURING REJECT *)
IF 	csp_case_transport_ls_trailing.axis.actual_position >330
	AND csp_case_transport_ls_trailing.axis.actual_position <355
THEN
	IF 	digital_input_is_active(case_present_os_di) 
		AND NOT temp1
	THEN
		bad_count_os :=  bad_count_os + 1;
		temp1 := TRUE;
	ELSE
		bad_count_os := 0;	
	END_IF
	
	IF 	digital_input_is_active(case_present_ls_di) 
		AND NOT temp2
	THEN
		bad_count_ls :=  bad_count_ls + 1;
		temp2 := TRUE;
	ELSE
		bad_count_ls := 0;	
	END_IF
END_IF

IF 	temp1 
	AND NOT digital_input_is_active(case_present_os_di)
THEN
	temp1 := FALSE;
END_IF

IF 	temp2 
	AND NOT digital_input_is_active(case_present_ls_di)
THEN
	temp2 := FALSE;
END_IF

IF (bad_count_os >= consecutive_blocked_count )
	AND
  (machine_is_stopped(csp.mch)
	OR machine_is_stop_emergency_active(csp.mch))
THEN
	bad_count_os := 0;
	process_message_reset(consecutive_blocked_os_aem);
END_IF

IF  process_message_is_on(consecutive_blocked_os_aem)
	AND
   (machine_is_stopped(csp.mch)
	OR
	machine_is_stop_emergency_active(csp.mch))
THEN
	bad_count_os := 0;	
	process_message_reset(consecutive_blocked_os_aem);
END_IF

IF bad_count_os >= consecutive_blocked_count
THEN
	process_message_set(1, 1, 1, consecutive_blocked_os_aem);
END_IF

IF (bad_count_ls >= consecutive_blocked_count )
	AND
	  (machine_is_stopped(csp.mch)
	OR 
	   machine_is_stop_emergency_active(csp.mch))
THEN
	bad_count_ls := 0;
	process_message_reset(consecutive_blocked_ls_aem);
END_IF

IF 	process_message_is_on(consecutive_blocked_ls_aem)
	AND
 	 (machine_is_stopped(csp.mch)
	OR 
	   machine_is_stop_emergency_active(csp.mch))
THEN
	bad_count_ls := 0;
	process_message_reset(consecutive_blocked_ls_aem);
END_IF

IF bad_count_ls >= consecutive_blocked_count
THEN
	process_message_set(1, 1, 1, consecutive_blocked_ls_aem);
END_IF

	
IF csp_case_main_services.dry_cycle_mode
	OR csp_main_motorization.empty_command
THEN
	check_section_disable(case_present_os_di_dchk);
	check_section_disable(case_present_ls_di_dchk);
ELSE
	check_section_enable(case_present_os_di_dchk);
	check_section_enable(case_present_ls_di_dchk);
END_IF			
(************************************************************************)

_handle_messages();

_write_output();

ACTION _handle_messages:
;
END_ACTION

ACTION _handle_process_test:
;
END_ACTION

ACTION _mode_manager:
IF process_mode_req_is_pending(prc)
THEN
    process_apply_mode_req_first_step(prc);
    CASE process_get_mode(prc) OF
        MODE_TO_ABSENT:
			;
        MODE_TO_INACTIVE:
			;
        MODE_TO_TEST:
			;
        MODE_TO_OPERATIONAL:
			;
    END_CASE
    process_apply_mode_req_second_step(prc);
END_IF
END_ACTION

ACTION _object_manager:
IF objects_initialization()
THEN
	sub_process_init(
		object_name					:= 'csp_case_glue_sensors.prc', 
		process						:= csp_case_glue.prc, 
		CONVERSION_this				:= prc);
		
	prc_path 						:= process_get_path(prc);
	
	(* INPUTS *)
	digital_input_init(
		object_name					:= CONCAT(prc_path, '_case_present_os_di'), 
		polarity_direct				:= TRUE, 
		process						:= prc, 
		CONVERSION_this				:= case_present_os_di);
		
digital_input_init(
		object_name					:= CONCAT(prc_path, '_case_present_ls_di'), 
		polarity_direct				:= TRUE, 
		process						:= prc, 
		CONVERSION_this				:= case_present_ls_di);
	
		
(* CHECK SECTION FOR THE OPERATOR SIDE GLUE PE SETS SHIFT REGISTER AND PE FAILURE LOGIC *)	
	check_section_window_mode_init(
		object_name:= CONCAT(prc_path, '_case_present_os_di_dchk'),
		check_enable:= TRUE, 
		event_to_check:= CHECK_SECTION_EVENT_INPUT_ON, 
		execution_mode:= CHECK_SECTION_EXECUTION_WHEN_EVENT_OCCURRED, 
		diagnostic_enable:= FALSE, 
		status_bits_to_be_true:= ITEM_CASE_FEED, 
		status_bits_to_be_false:= common_global_variables.NONE, 
		_step_status_conditioning_execution:= FALSE, 
		status_bits_to_set:= ITEM_HAS_OS_UPPER_FLAP_AT_GLUE, 
		status_bits_to_reset:=common_global_variables.NONE, 
		reject_bit_to_set:= 0, 
		_step:= 27, 
		first_step_to_write_offset:= 0, 
		number_of_steps_to_write:= 1, 
		begin_phase:= Case_at_glue_begin_phase,
		end_phase:= Case_at_glue_end_phase,
		max_consecutive_failed_checks:= 3, 
		max_failed_checks_percentage:= 100, 
		products_for_failed_checks_percentage:= 100, 
		shift_register:= csp_case_main_statistics.sr , 
		process:= prc, 
		CONVERSION_this:= case_present_os_di_dchk );

	check_section_add_di_input(
		di_input := case_present_os_di,
		CONVERSION_this:= case_present_os_di_dchk);
	 	
(* CHECK SECTION FOR THE LOADER SIDE GLUE PE SETS SHIFT REGISTER AND PE FAILURE LOGIC *)	
	check_section_window_mode_init(
		object_name:= CONCAT(prc_path, '_case_present_ls_di_dchk'),
		check_enable:= TRUE, 
		event_to_check:= CHECK_SECTION_EVENT_INPUT_ON, 
		execution_mode:= CHECK_SECTION_EXECUTION_WHEN_EVENT_OCCURRED, 
		diagnostic_enable:= FALSE, 
		status_bits_to_be_true:= ITEM_CASE_FEED, 
		status_bits_to_be_false:= common_global_variables.NONE, 
		_step_status_conditioning_execution:= FALSE, 
		status_bits_to_set:= ITEM_HAS_LS_UPPER_FLAP_AT_GLUE, 
		status_bits_to_reset:= common_global_variables.NONE, 
		reject_bit_to_set:= 0, 
		_step:= 27, 
		first_step_to_write_offset:= 0, 
		number_of_steps_to_write:= 1, 
		begin_phase:= Case_at_glue_begin_phase,
		end_phase:= Case_at_glue_end_phase,
		max_consecutive_failed_checks:= 3, 
		max_failed_checks_percentage:= 100, 
		products_for_failed_checks_percentage:= 100, 
		shift_register:= csp_case_main_statistics.sr , 
		process:= prc, 
		CONVERSION_this:= case_present_ls_di_dchk );

	check_section_add_di_input(
		di_input := case_present_ls_di,
		CONVERSION_this:= case_present_ls_di_dchk);
	
	process_message_init(
		object_name:= CONCAT(prc_path, '_consecutive_blocked_os_aem'), 
		behaviour:= MESSAGE_BEHAVIOUR_STATE, 
		reset_timeout:= 0, 
		disableable:= FALSE, 
		individual_reset:= FALSE, 
		machine_reaction:= MACHINE_REACTION_STOP_IN_PHASE_ONE, 
		typology:= MESSAGE_TYPOLOGY_ABNORMAL, 
		process:= prc, 
		CONVERSION_this:= consecutive_blocked_os_aem);
	
	process_message_init(
		object_name:= CONCAT(prc_path, '_consecutive_blocked_ls_aem'), 
		behaviour:= MESSAGE_BEHAVIOUR_STATE, 
		reset_timeout:= 0, 
		disableable:= FALSE, 
		individual_reset:= FALSE, 
		machine_reaction:= MACHINE_REACTION_STOP_IN_PHASE_ONE, 
		typology:= MESSAGE_TYPOLOGY_ABNORMAL, 
		process:= prc, 
		CONVERSION_this:= consecutive_blocked_ls_aem);
	
		
END_IF

IF objects_running()
THEN
	process_cycle(prc);
	
END_IF
END_ACTION

ACTION _read_process_image:
;
END_ACTION

ACTION _read_var_input:
;
END_ACTION

ACTION _set_runtime_properties:
;
END_ACTION

ACTION _write_output:
;
END_ACTION

END_PROGRAM

// ---- Tools/Common/csp_interface_configuration.TcPOU
FUNCTION csp_interface_configuration : VOID
VAR_IN_OUT
	motman:																motorization_manager;
	machine:															machine;
	
	CONVERSION_this:													csp_main_configurator_struct;			
END_VAR

CONVERSION_this.motman_ref																:= ADR(motman);
CONVERSION_this.machine_ref																:= ADR(machine);

END_FUNCTION

// ---- Application/CSP/Case/_Tasks/_csp_case_highest.TcPOU
(*********************************** G.D S.p.A. - Technical Department ***********************************
============= PROGRAM INFO ============
FOLDER:             TBD
MACHINES INVOLVED:  TBD 

============= DESCRIPTION =============
csp main interface program

============= REVISIONS ===============
Date		Version	 	Author      	Description             
----------	-------		------------  	--------------------------------------------
2019/09/27 	0000.00	 	M.Grasso		Creation of the PRG

**********************************************************************************************************)
PROGRAM _csp_case_highest
VAR
END_VAR

csp_case_virtualMaster();

_csp_case_closing_highest();

_csp_case_discharge_highest();

_csp_case_feed_highest();

_csp_case_flapControl_highest();

_csp_case_glue_highest();

_csp_case_loader_highest();

_csp_case_openFlap_highest();

_csp_case_main_highest();

_csp_case_topRail_highest();

_csp_case_transport_highest();

END_PROGRAM

// ---- Application/CSP/Case/Closing/_Tasks/_csp_case_closing_highest.TcPOU
(*********************************** G.D S.p.A. - Technical Department ***********************************
============= PROGRAM INFO ============
FOLDER:             TBD
MACHINES INVOLVED:  TBD 

============= DESCRIPTION =============
csp main interface program

============= REVISIONS ===============
Date		Version	 	Author      	Description             
----------	-------		------------  	--------------------------------------------
2019/09/27 	0000.00	 	M.Grasso		Creation of the PRG

**********************************************************************************************************)
PROGRAM _csp_case_closing_highest
VAR
END_VAR

csp_case_closing();

(* CASE *)
	(* CLOSING *)
		(* OS *)
		csp_case_closing_os_horizontal();
		csp_case_closing_os_upper();
		csp_case_closing_os_lower();
	
		(* LS *)
		csp_case_closing_ls_horizontal();
		csp_case_closing_ls_upper();
		csp_case_closing_ls_lower();

END_PROGRAM

// ---- Application/CSP/Case/Discharge/_Tasks/_csp_case_discharge_highest.TcPOU
(*********************************** G.D S.p.A. - Technical Department ***********************************
============= PROGRAM INFO ============
FOLDER:             TBD
MACHINES INVOLVED:  TBD 

============= DESCRIPTION =============
csp main interface program

============= REVISIONS ===============
Date		Version	 	Author      	Description             
----------	-------		------------  	--------------------------------------------
2019/09/27 	0000.00	 	M.Grasso		Creation of the PRG

**********************************************************************************************************)
PROGRAM _csp_case_discharge_highest
VAR
END_VAR

csp_case_discharge();

END_PROGRAM

// ---- Application/CSP/Case/Discharge/csp_case_discharge.TcPOU
(*********************************** G.D S.p.A. - Technical Department ***********************************
============= PROGRAM INFO ============
FOLDER:             TBD
MACHINES INVOLVED:  TBD 

============= DESCRIPTION =============
csp machine declaration

============= REVISIONS ===============
Date		Version	 	Author      	Description             
----------	-------		------------  	--------------------------------------------
2019/04/05 	0000.00	 	M.Grasso		Creation of the PRG

**********************************************************************************************************)
(*$R process_ref := prc; $*)
PROGRAM csp_case_discharge
VAR
		
	prc:											process;
	prc_path:										STRING;
	
END_VAR

_read_var_input();

_object_manager();

IF NOT objects_running()
THEN
	RETURN;	
END_IF

_read_process_image();

_mode_manager();

_set_runtime_properties();

(********************************* BODY *********************************)
(************************************************************************)

_handle_messages();

_write_output();

ACTION _handle_messages:
;
END_ACTION

ACTION _handle_process_test:
;
END_ACTION

ACTION _mode_manager:
IF process_mode_req_is_pending(prc)
THEN
    process_apply_mode_req_first_step(prc);
    CASE process_get_mode(prc) OF
        MODE_TO_ABSENT:
			;
        MODE_TO_INACTIVE:
			;
        MODE_TO_TEST:
			;
        MODE_TO_OPERATIONAL:
			;
    END_CASE
    process_apply_mode_req_second_step(prc);
END_IF
END_ACTION

ACTION _object_manager:
IF objects_initialization()
THEN
	sub_process_init(
		object_name					:= 'csp_case_discharge.prc', 
		process						:= csp_case.prc, 
		CONVERSION_this				:= prc);
		
	prc_path 						:= process_get_path(prc);
END_IF

IF objects_running()
THEN
	process_cycle(prc);
END_IF
END_ACTION

ACTION _read_process_image:
;
END_ACTION

ACTION _read_var_input:
;
END_ACTION

ACTION _set_runtime_properties:
;
END_ACTION

ACTION _write_output:
;
END_ACTION

END_PROGRAM

// ---- Application/CSP/Case/Feed/_Tasks/_csp_case_feed_highest.TcPOU
(*********************************** G.D S.p.A. - Technical Department ***********************************
============= PROGRAM INFO ============
FOLDER:             TBD
MACHINES INVOLVED:  TBD 

============= DESCRIPTION =============
csp main interface program

============= REVISIONS ===============
Date		Version	 	Author      	Description             
----------	-------		------------  	--------------------------------------------
2019/09/27 	0000.00	 	M.Grasso		Creation of the PRG

**********************************************************************************************************)
PROGRAM _csp_case_feed_highest
VAR
END_VAR

csp_case_feed();

(* CASE *)
	(* FEED *)
		(* ARM *)
		csp_case_feed_arm_elbow();
		csp_case_feed_arm_sensors();
		csp_case_feed_arm_shoulder();
		csp_case_feed_arm_wrist();
		csp_case_feed_kinematic();
			csp_case_feed_kinematic_x();
			csp_case_feed_kinematic_y();
			csp_case_feed_kinematic_tilt();
		csp_case_feed_virtualMaster();
		
	(* SHUTTLE *)
			(* HORIZONTAL *)
			csp_case_feed_shuttle_horizontal();
			(* SENSORS *)
			csp_case_feed_shuttle_sensors();
			csp_case_feed_shuttle_sensors_os();
			csp_case_feed_shuttle_sensors_ls();
			(*VERTICAL*)
			csp_case_feed_shuttle_vertical();

END_PROGRAM

// ---- Application/CSP/Case/Flap Control/_Tasks/_csp_case_flapControl_highest.TcPOU
(*********************************** G.D S.p.A. - Technical Department ***********************************
============= PROGRAM INFO ============
FOLDER:             TBD
MACHINES INVOLVED:  TBD 

============= DESCRIPTION =============
csp main interface program

============= REVISIONS ===============
Date		Version	 	Author      	Description             
----------	-------		------------  	--------------------------------------------
2019/09/27 	0000.00	 	M.Grasso		Creation of the PRG

**********************************************************************************************************)
PROGRAM _csp_case_flapControl_highest
VAR
END_VAR

csp_case_flapControl();


		(* LS *)
		(* UPPER *)
			csp_case_fc_ls_upper();
			csp_case_fc_ls_upper_follower();
			csp_case_fc_ls_upper_sensors();
			csp_case_fc_ls_upper_leadingMinorCloser();
			csp_case_fc_ls_upper_leadingMinorCloser_virtual();
			csp_case_fc_ls_upper_spreader();
			(* LOWER *)
			csp_case_fc_ls_lower();
			csp_case_fc_ls_lower_follower();
			csp_case_fc_ls_lower_sensors();
			csp_case_fc_ls_lower_spreader();
			csp_case_fc_ls_lower_trailingCloser();
		(* OS *)
			(* UPPER *)
			csp_case_fc_os_upper();
			csp_case_fc_os_upper_follower();
			csp_case_fc_os_upper_sensors();
			csp_case_fc_os_upper_spreader();
			(* LOWER *)
			csp_case_fc_os_lower();
			csp_case_fc_os_lower_follower();
			csp_case_fc_os_lower_sensors();
			csp_case_fc_os_lower_spreader();

END_PROGRAM

// ---- Application/CSP/Case/Glue/_Tasks/_csp_case_glue_highest.TcPOU
(*********************************** G.D S.p.A. - Technical Department ***********************************
============= PROGRAM INFO ============
FOLDER:             TBD
MACHINES INVOLVED:  TBD 

============= DESCRIPTION =============
csp main interface program

============= REVISIONS ===============
Date		Version	 	Author      	Description             
----------	-------		------------  	--------------------------------------------
2019/09/27 	0000.00	 	M.Grasso		Creation of the PRG

**********************************************************************************************************)
PROGRAM _csp_case_glue_highest
VAR
END_VAR

csp_case_glue();
csp_case_glue_hotMelt();


(* CASE *)
	(* GLUE *)
		(* LS *)
			(* GUNS *)
			csp_case_glue_ls_guns();
		(* OS *)
			(* ACC-U-CHANGE*)
			(* GUNS *)
			csp_case_glue_os_guns();
		
		(* SENSORS *)
		csp_case_glue_sensors();

END_PROGRAM

// ---- Application/CSP/Case/Loader/_Tasks/_csp_case_loader_highest.TcPOU
 (*********************************** G.D S.p.A. - Technical Department ***********************************
============= PROGRAM INFO ============
FOLDER:             TBD
MACHINES INVOLVED:  TBD 

============= DESCRIPTION =============
csp main interface program

============= REVISIONS ===============
Date		Version	 	Author      	Description             
----------	-------		------------  	--------------------------------------------
2019/09/27 	0000.00	 	M.Grasso		Creation of the PRG

**********************************************************************************************************)
PROGRAM _csp_case_loader_highest
VAR
END_VAR

csp_case_loader();

(* CASE *)
	(* LOADER *)
		(* PUSHER *)
		csp_case_loader_pusher();
		(* SENSORS *)
		csp_case_loader_virtualMaster();

END_PROGRAM

// ---- Application/CSP/Case/Open Flap/_Tasks/_csp_case_openFlap_highest.TcPOU
(*********************************** G.D S.p.A. - Technical Department ***********************************
============= PROGRAM INFO ============
FOLDER:             TBD
MACHINES INVOLVED:  TBD 

============= DESCRIPTION =============
csp main interface program

============= REVISIONS ===============
Date		Version	 	Author      	Description             
----------	-------		------------  	--------------------------------------------
2019/09/27 	0000.00	 	M.Grasso		Creation of the PRG

**********************************************************************************************************)
PROGRAM _csp_case_openFlap_highest
VAR
END_VAR

csp_case_openFlap();

END_PROGRAM

// ---- Application/CSP/Case/Open Flap/csp_case_openFlap.TcPOU
(*********************************** G.D S.p.A. - Technical Department ***********************************
============= PROGRAM INFO ============
FOLDER:             TBD
MACHINES INVOLVED:  TBD 

============= DESCRIPTION =============
csp machine declaration

============= REVISIONS ===============
Date		Version	 	Author      	Description             
----------	-------		------------  	--------------------------------------------
2019/04/05 	0000.00	 	M.Grasso		Creation of the PRG

**********************************************************************************************************)
(*$R process_ref := prc; $*)
PROGRAM csp_case_openFlap
VAR
	
	prc:											process;
	prc_path:										STRING;
	
END_VAR

_read_var_input();

_object_manager();

IF NOT objects_running()
THEN
	RETURN;	
END_IF

_read_process_image();

_mode_manager();

_set_runtime_properties();

(********************************* BODY *********************************)
(************************************************************************)

_handle_messages();

_write_output();

ACTION _handle_messages:
;
END_ACTION

ACTION _handle_process_test:
;
END_ACTION

ACTION _mode_manager:
IF process_mode_req_is_pending(prc)
THEN
    process_apply_mode_req_first_step(prc);
    CASE process_get_mode(prc) OF
        MODE_TO_ABSENT:
			;
        MODE_TO_INACTIVE:
			;
        MODE_TO_TEST:
			;
        MODE_TO_OPERATIONAL:
			;
    END_CASE
    process_apply_mode_req_second_step(prc);
END_IF
END_ACTION

ACTION _object_manager:
IF objects_initialization()
THEN
	sub_process_init(
		object_name					:= 'csp_case_openFlap.prc', 
		process						:= csp_case.prc, 
		CONVERSION_this				:= prc);
		
	prc_path 						:= process_get_path(prc);
END_IF

IF objects_running()
THEN
	process_cycle(prc);
END_IF
END_ACTION

ACTION _read_process_image:
;
END_ACTION

ACTION _read_var_input:
;
END_ACTION

ACTION _set_runtime_properties:
;
END_ACTION

ACTION _write_output:
;
END_ACTION

END_PROGRAM

// ---- Application/CSP/Case/Main/_Tasks/_csp_case_main_highest.TcPOU
(*********************************** G.D S.p.A. - Technical Department ***********************************
============= PROGRAM INFO ============
FOLDER:             TBD
MACHINES INVOLVED:  TBD 

============= DESCRIPTION =============
csp main interface program

============= REVISIONS ===============
Date		Version	 	Author      	Description             
----------	-------		------------  	--------------------------------------------
2019/09/27 	0000.00	 	M.Grasso		Creation of the PRG

**********************************************************************************************************)
PROGRAM _csp_case_main_highest
VAR
END_VAR

csp_case_main_statistics();
csp_case_main_statistics_debug();

END_PROGRAM

// ---- Application/CSP/Case/Main/statistics/csp_case_main_statistics_debug.TcPOU
(*$R
    process_ref:= csp_case_main_statistics.prc;
$*)
PROGRAM csp_case_main_statistics_debug
VAR
	step_id:							INT;

	outer_shift_debug:					ARRAY[0..STEP_ARRAY_UPPER_INDEX] OF csp_case_main_statistics_debug_struct;
	outer_shift_register_step_pointer:	POINTER TO shift_register_step_type;
	
END_VAR

IF 	NOT objects_running()
THEN
	RETURN;
END_IF

(*======================== PROGRAM HANDLER ===========================*)


FOR step_id:= 1 TO 30 BY 1 DO
	outer_shift_debug[step_id].step_id:= step_id;
 	outer_shift_register_step_pointer:= shift_register_read_step(step_id, csp_case_main_statistics.sr);
	outer_shift_debug[step_id].status:= outer_shift_register_step_pointer^.status;
	outer_shift_debug[step_id].reject_reason:= outer_shift_register_step_pointer^.first_reject_info.reason;
	//outer_shift_debug[step_id].item_has := outer_shift_register_step_pointer^.

	
END_FOR 
IF step_id = 31//csp_case_main_statistics.SHIFT_LAST_STEP +1
	THEN
	step_id  :=1;
END_IF

END_PROGRAM

// ---- Application/CSP/Case/Top Rail/_Tasks/_csp_case_topRail_highest.TcPOU
(*********************************** G.D S.p.A. - Technical Department ***********************************
============= PROGRAM INFO ============
FOLDER:             TBD
MACHINES INVOLVED:  TBD 

============= DESCRIPTION =============
csp main interface program

============= REVISIONS ===============
Date		Version	 	Author      	Description             
----------	-------		------------  	--------------------------------------------
2019/09/27 	0000.00	 	M.Grasso		Creation of the PRG

**********************************************************************************************************)
PROGRAM _csp_case_topRail_highest
VAR
END_VAR

csp_case_topRail();

(* CASE *)
	(* TOP RAIL *)
		(* SQUARING *)
		csp_case_topRail_squaring();

END_PROGRAM

// ---- Application/CSP/Case/Top Rail/csp_case_topRail.TcPOU
(*********************************** G.D S.p.A. - Technical Department ***********************************
============= PROGRAM INFO ============
FOLDER:             TBD
MACHINES INVOLVED:  TBD 

============= DESCRIPTION =============
csp machine declaration

============= REVISIONS ===============
Date		Version	 	Author      	Description             
----------	-------		------------  	--------------------------------------------
2019/04/05 	0000.00	 	M.Grasso		Creation of the PRG

**********************************************************************************************************)
(*$R process_ref := prc; $*)
PROGRAM csp_case_topRail
VAR
	
	prc:											process;
	prc_path:										STRING;
	
END_VAR

_read_var_input();

_object_manager();

IF NOT objects_running()
THEN
	RETURN;	
END_IF

_read_process_image();

_mode_manager();

_set_runtime_properties();

(********************************* BODY *********************************)
(************************************************************************)

_handle_messages();

_write_output();

ACTION _handle_messages:
;
END_ACTION

ACTION _handle_process_test:
;
END_ACTION

ACTION _mode_manager:
IF process_mode_req_is_pending(prc)
THEN
    process_apply_mode_req_first_step(prc);
    CASE process_get_mode(prc) OF
        MODE_TO_ABSENT:
			;
        MODE_TO_INACTIVE:
			;
        MODE_TO_TEST:
			;
        MODE_TO_OPERATIONAL:
			;
    END_CASE
    process_apply_mode_req_second_step(prc);
END_IF
END_ACTION

ACTION _object_manager:
IF objects_initialization()
THEN
	sub_process_init(
		object_name					:= 'csp_case_topRail.prc', 
		process						:= csp_case.prc, 
		CONVERSION_this				:= prc);
		
	prc_path 						:= process_get_path(prc);
END_IF

IF objects_running()
THEN
	process_cycle(prc);
END_IF
END_ACTION

ACTION _read_process_image:
;
END_ACTION

ACTION _read_var_input:
;
END_ACTION

ACTION _set_runtime_properties:
;
END_ACTION

ACTION _write_output:
;
END_ACTION

END_PROGRAM

// ---- Application/CSP/Case/Top Rail/Squaring/csp_case_topRail_squaring.TcPOU
(*********************************** G.D S.p.A. - Technical Department ***********************************
============= PROGRAM INFO ============
FOLDER:             TBD
MACHINES INVOLVED:  TBD 

============= DESCRIPTION =============
csp machine declaration

============= REVISIONS ===============
Date		Version	 	Author      	Description             
----------	-------		------------  	--------------------------------------------
2019/04/05 	0000.00	 	M.Grasso		Creation of the PRG

**********************************************************************************************************)
(*$R process_ref := prc; $*)
PROGRAM csp_case_topRail_squaring
VAR
	
	prc:											process;
	prc_path:										STRING;
	
END_VAR

_read_var_input();

_object_manager();

IF NOT objects_running()
THEN
	RETURN;	
END_IF

_read_process_image();

_mode_manager();

_set_runtime_properties();

(********************************* BODY *********************************)
(************************************************************************)

_handle_messages();

_write_output();

ACTION _handle_messages:
;
END_ACTION

ACTION _handle_process_test:
;
END_ACTION

ACTION _mode_manager:
IF process_mode_req_is_pending(prc)
THEN
    process_apply_mode_req_first_step(prc);
    CASE process_get_mode(prc) OF
        MODE_TO_ABSENT:
			;
        MODE_TO_INACTIVE:
			;
        MODE_TO_TEST:
			;
        MODE_TO_OPERATIONAL:
			;
    END_CASE
    process_apply_mode_req_second_step(prc);
END_IF
END_ACTION

ACTION _object_manager:
IF objects_initialization()
THEN
	sub_process_init(
		object_name					:= 'csp_case_topRail_squaring.prc', 
		process						:= csp_case_topRail.prc, 
		CONVERSION_this				:= prc);
		
	prc_path 						:= process_get_path(prc);
END_IF

IF objects_running()
THEN
	process_cycle(prc);
END_IF
END_ACTION

ACTION _read_process_image:
;
END_ACTION

ACTION _read_var_input:
;
END_ACTION

ACTION _set_runtime_properties:
;
END_ACTION

ACTION _write_output:
;
END_ACTION

END_PROGRAM

// ---- Application/CSP/Case/Transport/_Tasks/_csp_case_transport_highest.TcPOU
(*********************************** G.D S.p.A. - Technical Department ***********************************
============= PROGRAM INFO ============
FOLDER:             TBD
MACHINES INVOLVED:  TBD 

============= DESCRIPTION =============
csp main interface program

============= REVISIONS ===============
Date		Version	 	Author      	Description             
----------	-------		------------  	--------------------------------------------
2019/09/27 	0000.00	 	M.Grasso		Creation of the PRG

**********************************************************************************************************)
PROGRAM _csp_case_transport_highest
VAR
END_VAR

csp_case_transport();
csp_case_transport_virtualMaster();

(* CSP *)
	(* TRANSPORT *)
		(* LS *)
		csp_case_transport_ls();
		(* OS *)
		csp_case_transport_os();
		
(* CSP *)
(* TRANSPORT *)
	(* LS *)
	csp_case_transport_ls_leading();
	csp_case_transport_ls_trailing();
	(* OS *)
	csp_case_transport_os_leading();
	csp_case_transport_os_trailing();
	(* TENSIONER *)
	;

END_PROGRAM

// ---- Application/CSP/Case/Transport/LS/csp_case_transport_ls.TcPOU
(*********************************** G.D S.p.A. - Technical Department ***********************************
============= PROGRAM INFO ============
FOLDER:             TBD
MACHINES INVOLVED:  TBD 

============= DESCRIPTION =============
csp machine declaration

============= REVISIONS ===============
Date		Version	 	Author      	Description             
----------	-------		------------  	--------------------------------------------
2019/04/05 	0000.00	 	M.Grasso		Creation of the PRG

**********************************************************************************************************)
(*$R process_ref := prc; $*)
PROGRAM csp_case_transport_ls
VAR
	
	prc:											process;
	prc_path:										STRING;
	
END_VAR

_read_var_input();

_object_manager();

IF NOT objects_running()
THEN
	RETURN;	
END_IF

_read_process_image();

_mode_manager();

_set_runtime_properties();

(********************************* BODY *********************************)
(************************************************************************)

_handle_messages();

_write_output();

ACTION _handle_messages:
;
END_ACTION

ACTION _handle_process_test:
;
END_ACTION

ACTION _mode_manager:
IF process_mode_req_is_pending(prc)
THEN
    process_apply_mode_req_first_step(prc);
    CASE process_get_mode(prc) OF
        MODE_TO_ABSENT:
			;
        MODE_TO_INACTIVE:
			;
        MODE_TO_TEST:
			;
        MODE_TO_OPERATIONAL:
			;
    END_CASE
    process_apply_mode_req_second_step(prc);
END_IF
END_ACTION

ACTION _object_manager:
IF objects_initialization()
THEN
	sub_process_init(
		object_name					:= 'csp_case_transport_ls.prc', 
		process						:= csp_case_transport.prc, 
		CONVERSION_this				:= prc);
		
	prc_path 						:= process_get_path(prc);
END_IF

IF objects_running()
THEN
	process_cycle(prc);
END_IF
END_ACTION

ACTION _read_process_image:
;
END_ACTION

ACTION _read_var_input:
;
END_ACTION

ACTION _set_runtime_properties:
;
END_ACTION

ACTION _write_output:
;
END_ACTION

END_PROGRAM

// ---- Application/CSP/Case/Transport/OS/csp_case_transport_os.TcPOU
(*********************************** G.D S.p.A. - Technical Department ***********************************
============= PROGRAM INFO ============
FOLDER:             TBD
MACHINES INVOLVED:  TBD 

============= DESCRIPTION =============
csp machine declaration

============= REVISIONS ===============
Date		Version	 	Author      	Description             
----------	-------		------------  	--------------------------------------------
2019/04/05 	0000.00	 	M.Grasso		Creation of the PRG

**********************************************************************************************************)
(*$R process_ref := prc; $*)
PROGRAM csp_case_transport_os
VAR
	
	prc:											process;
	prc_path:										STRING;
	
END_VAR

_read_var_input();

_object_manager();

IF NOT objects_running()
THEN
	RETURN;	
END_IF

_read_process_image();

_mode_manager();

_set_runtime_properties();

(********************************* BODY *********************************)
(************************************************************************)

_handle_messages();

_write_output();

ACTION _handle_messages:
;
END_ACTION

ACTION _handle_process_test:
;
END_ACTION

ACTION _mode_manager:
IF process_mode_req_is_pending(prc)
THEN
    process_apply_mode_req_first_step(prc);
    CASE process_get_mode(prc) OF
        MODE_TO_ABSENT:
			;
        MODE_TO_INACTIVE:
			;
        MODE_TO_TEST:
			;
        MODE_TO_OPERATIONAL:
			;
    END_CASE
    process_apply_mode_req_second_step(prc);
END_IF
END_ACTION

ACTION _object_manager:
IF objects_initialization()
THEN
	sub_process_init(
		object_name					:= 'csp_case_transport_os.prc', 
		process						:= csp_case_transport.prc, 
		CONVERSION_this				:= prc);
		
	prc_path 						:= process_get_path(prc);
END_IF

IF objects_running()
THEN
	process_cycle(prc);
END_IF
END_ACTION

ACTION _read_process_image:
;
END_ACTION

ACTION _read_var_input:
;
END_ACTION

ACTION _set_runtime_properties:
;
END_ACTION

ACTION _write_output:
;
END_ACTION

END_PROGRAM

// ---- Application/CSP/Transfer/_Tasks/_csp_transfer_highest.TcPOU
(*********************************** G.D S.p.A. - Technical Department ***********************************
============= PROGRAM INFO ============
FOLDER:             TBD
MACHINES INVOLVED:  TBD 

============= DESCRIPTION =============
csp main interface program

============= REVISIONS ===============
Date		Version	 	Author      	Description             
----------	-------		------------  	--------------------------------------------
2019/09/27 	0000.00	 	M.Grasso		Creation of the PRG

**********************************************************************************************************)
PROGRAM _csp_transfer_highest
VAR
END_VAR

csp_transfer();

(* SWAPPED CROSSPUSHER AND ACCUMULATOR BECAUSE ACCUMULATOR LOOKS AT CROSSPUSHER NEXT CAM *)



_csp_transfer_upstacker_highest();


_csp_transfer_crosspusher_highest();

_csp_transfer_accumulator_highest();


_csp_transfer_main_highest();

_csp_transfer_infeed_highest();

csp_transfer_virtualMaster();

END_PROGRAM

// ---- Application/CSP/Transfer/Accumulator/_Tasks/_csp_transfer_accumulator_highest.TcPOU
(*********************************** G.D S.p.A. - Technical Department ***********************************
============= PROGRAM INFO ============
FOLDER:             TBD
MACHINES INVOLVED:  TBD 

============= DESCRIPTION =============
csp main interface program

============= REVISIONS ===============
Date		Version	 	Author      	Description             
----------	-------		------------  	--------------------------------------------
2019/09/27 	0000.00	 	M.Grasso		Creation of the PRG

**********************************************************************************************************)
PROGRAM _csp_transfer_accumulator_highest
VAR
END_VAR

csp_transfer_accumulator();
(* TRANSFER *)
	(* ACCUMULATOR *)
		(* ACCU-U-CHANGE*)
		csp_transfer_accumulator_accU();
		(* FINGER *)
		csp_transfer_accumulator_finger();
		(* LIFT *)
		csp_transfer_accumulator_lift();
		(* BELT *)
		csp_transfer_accumulator_virtualMaster();
		csp_transfer_accumulator_belt();

END_PROGRAM

// ---- Application/CSP/Transfer/Accumulator/Acc U Change/csp_transfer_accumulator_accU.TcPOU
(*********************************** G.D S.p.A. - Technical Department ***********************************
============= PROGRAM INFO ============
FOLDER:             TBD
MACHINES INVOLVED:  TBD 

============= DESCRIPTION =============
csp machine declaration

============= REVISIONS ===============
Date		Version	 	Author      	Description             
----------	-------		------------  	--------------------------------------------
2019/04/05 	0000.00	 	M.Grasso		Creation of the PRG

**********************************************************************************************************)
(*$R process_ref := prc; $*)
PROGRAM csp_transfer_accumulator_accU
VAR
	
	prc:											process;
	prc_path:										STRING;
	
END_VAR

_read_var_input();

_object_manager();

IF NOT objects_running()
THEN
	RETURN;	
END_IF

_read_process_image();

_mode_manager();

_set_runtime_properties();

(********************************* BODY *********************************)
(************************************************************************)

_handle_messages();

_write_output();

ACTION _handle_messages:
;
END_ACTION

ACTION _handle_process_test:
;
END_ACTION

ACTION _mode_manager:
IF process_mode_req_is_pending(prc)
THEN
    process_apply_mode_req_first_step(prc);
    CASE process_get_mode(prc) OF
        MODE_TO_ABSENT:
			;
        MODE_TO_INACTIVE:
			;
        MODE_TO_TEST:
			;
        MODE_TO_OPERATIONAL:
			;
    END_CASE
    process_apply_mode_req_second_step(prc);
END_IF
END_ACTION

ACTION _object_manager:
IF objects_initialization()
THEN
	sub_process_init(
		object_name					:= 'csp_transfer_accumulator_accU.prc', 
		process						:= csp_transfer_accumulator.prc, 
		CONVERSION_this				:= prc);
		
	prc_path 						:= process_get_path(prc);
END_IF

IF objects_running()
THEN
	process_cycle(prc);
END_IF
END_ACTION

ACTION _read_process_image:
;
END_ACTION

ACTION _read_var_input:
;
END_ACTION

ACTION _set_runtime_properties:
;
END_ACTION

ACTION _write_output:
;
END_ACTION

END_PROGRAM

// ---- Application/CSP/Transfer/Accumulator/Finger/csp_transfer_accumulator_finger.TcPOU
(*********************************** G.D S.p.A. - Technical Department ***********************************
============= PROGRAM INFO ============
FOLDER:             TBD
MACHINES INVOLVED:  TBD 

============= DESCRIPTION =============
csp machine declaration

============= REVISIONS ===============
Date		Version	 	Author      	Description             
----------	-------		------------  	--------------------------------------------
2019/04/05 	0000.00	 	M.Grasso		Creation of the PRG

**********************************************************************************************************)
(*$R process_ref := prc; $*)
PROGRAM csp_transfer_accumulator_finger
VAR
	
	prc:											process;
	prc_path:										STRING;
	
	cam_id: INT;
END_VAR

_read_var_input();

_object_manager();

IF NOT objects_running()
THEN
	RETURN;	
END_IF

_read_process_image();

_mode_manager();

_set_runtime_properties();

(********************************* BODY *********************************)
IF csp_main_brand.count = '48Count'
	THEN
		cam_id := 39;
ELSE 
	cam_id := 34;
END_IF
(************************************************************************)

_handle_messages();

_write_output();

ACTION _handle_messages:
;
END_ACTION

ACTION _handle_process_test:
;
END_ACTION

ACTION _mode_manager:
IF process_mode_req_is_pending(prc)
THEN
    process_apply_mode_req_first_step(prc);
    CASE process_get_mode(prc) OF
        MODE_TO_ABSENT:
			;
        MODE_TO_INACTIVE:
			;
        MODE_TO_TEST:
			;
        MODE_TO_OPERATIONAL:
			;
    END_CASE
    process_apply_mode_req_second_step(prc);
END_IF
END_ACTION

ACTION _object_manager:
IF objects_initialization()
THEN
	sub_process_init(
		object_name					:= 'csp_transfer_accumulator_finger.prc', 
		process						:= csp_transfer_accumulator.prc, 
		CONVERSION_this				:= prc);
		
	prc_path 						:= process_get_path(prc);
END_IF

IF objects_running()
THEN
	process_cycle(prc);
END_IF
END_ACTION

ACTION _read_process_image:
;
END_ACTION

ACTION _read_var_input:
;
END_ACTION

ACTION _set_runtime_properties:
;
END_ACTION

ACTION _write_output:
;
END_ACTION

END_PROGRAM

// ---- Application/CSP/Transfer/Accumulator/Lift/csp_transfer_accumulator_lift.TcPOU
(*********************************** G.D S.p.A. - Technical Department ***********************************
============= PROGRAM INFO ============
FOLDER:             TBD
MACHINES INVOLVED:  TBD 

============= DESCRIPTION =============
csp machine declaration

============= REVISIONS ===============
Date		Version	 	Author      	Description             
----------	-------		------------  	--------------------------------------------
2019/04/05 	0000.00	 	M.Grasso		Creation of the PRG

**********************************************************************************************************)
(*$R process_ref := prc; $*)
PROGRAM csp_transfer_accumulator_lift
VAR
	
	prc:												process;
	prc_path:											STRING;
	
	fsm_enable_condition:								BOOL := FALSE;
	fsm_next_status:									CSP_TRANSFER_ACCUMULATOR_LIFT_STATUS_enum;
	fsm_status:											CSP_TRANSFER_ACCUMULATOR_LIFT_STATUS_enum;
	
	axis:												axis;
	phase_position_deg:									LREAL := 0;
	phase_velocity_degps:								LREAL := 100.0;
		
	home_position_master_offset_deg:					LREAL := 0.0;
	axis_calculate_cam_slave_master_position_deg:		LREAL := 0.0;
	axis_calculated_cam_slave_position_deg:				LREAL := 0.0;	
	slave_position_has_been_calculated:					BOOL  := FALSE;
	
	phase_enable:										BOOL := TRUE;
	slave_position_request:								BOOL := TRUE;
	engage_enable:										BOOL := TRUE;
	
	cam_id:												DINT ;
	slave_scaling:										LREAL := 1 (*360.0*);
	master_scaling:										LREAL := 1 (*360.0*);
	master_position:									LREAL := 30;
	master_cam:											LREAL := 30;
	
	master_offset:										LREAL := 0;
	master_offset_phase:								LREAL;
	master_engage_mode:									axis_cam_engage_mode_enum;
	slave_offset:										LREAL := 0;
	
	run:												BOOL;
	dwell:												BOOL;
	
	run_test:											BOOL;
	dwell_test:											BOOL;
	
	active_cam:											DINT := DWELL_CAM;
	next_cam:											DINT := DWELL_CAM;
	
	connection_status: 									csp_transfer_crosspusher_connection_status_enum;
	connection_status_next: 							csp_transfer_crosspusher_connection_status_enum;
	connection_done: 									BOOL;
	connection_running: 								BOOL;
	connection_error:									BOOL;
	connection_time_out_tmr:							timer;
	connection_faulted_aem:	 							message;
	connection_conditions:								BOOL;
	connection_done_motcond:							motorization_conditioner;
	connection_motorization_moving:						BOOL;
	
	next_activation_position:							LREAL;	
	activation_position:								LREAL := 0.0;
	
	
	phase_status: 										csp_transfer_crosspusher_phase_status_enum;
	phase_status_next: 									csp_transfer_crosspusher_phase_status_enum;
	phase_done: 										BOOL;
	phase_running: 										BOOL;
	phase_error:										BOOL;
	phase_time_out_tmr:									timer;
	phase_faulted_aem:	 								message;
	phase_conditions:									BOOL;
	phase_slave_position:								LREAL;
	
	
	disable_req:										BOOL;
	debug_state_machine:								BOOL := FALSE;
	debug_phase_machine_one_step:						BOOL := FALSE;
	debug_connection_machine_one_step:					BOOL := FALSE;
	debug_immediate_stop_aem:							message;
	debug_immediate_stop:								BOOL;

	torque_limit:										INT := 500; (*$P $*)
	torque_limit_old:									INT;	
	
	servo_on_condition: 								BOOL;
	enable_delay: TON;
	Torque_force_constant: 								LREAL := 0.98;
END_VAR

VAR CONSTANT
	MOTOR_MAX_VELOCITY_DEGPS:							LREAL := 9600;
	MOTOR_MAX_ACCELLERATION_DEGPS2:						LREAL := 4800;
	MOTOR_MAX_DECELLERATION_DEGPS2:						LREAL := 4800;
	MOTOR_MAX_JERK_DEGPS3:								LREAL := 100000000; 
	MOTOR_MAX_FOLLOWING_ERROR_DEG:						LREAL := 2;
END_VAR

_read_var_input();

_object_manager();

IF NOT objects_running()
THEN
	RETURN;	
END_IF

_read_process_image();

